LIN {X 0,Y 516.64,Z 251.361,A -85,B 0,C 180,E1 -4935.827,E2 -4935.827} C_VEL
LIN {X 0,Y 516.583,Z 256.504,A -85,B 0,C 180,E1 -4939.02,E2 -4939.02} C_VEL
LIN {X 0,Y 516.522,Z 261.674,A -85,B 0,C 180,E1 -4942.18,E2 -4942.18} C_VEL
LIN {X 0,Y 516.438,Z 265.584,A -85,B 0,C 180,E1 -4944.534,E2 -4944.534} C_VEL
LIN {X 0,Y 516.408,Z 269.551,A -85,B 0,C 180,E1 -4946.879,E2 -4946.879} C_VEL
LIN {X 0,Y 516.319,Z 273.421,A -85,B 0,C 180,E1 -4949.171,E2 -4949.171} C_VEL
LIN {X 0,Y 518.475,Z 285.209,A -85,B 0,C 180,E1 -4949.539,E2 -4949.539} C_VEL
LIN {X 0,Y 518.209,Z 297.677,A -85,B 0,C 180,E1 -4950,E2 -4950} C_VEL
LIN {X 0,Y 517.936,Z 309.297,A -85,B 0,C 180,E1 -4950.583,E2 -4950.583} C_VEL
LIN {X 0,Y 517.653,Z 319.894,A -85,B 0,C 180,E1 -4951.264,E2 -4951.264} C_VEL
LIN {X 0,Y 517.351,Z 330.743,A -85,B 0,C 180,E1 -4952.141,E2 -4952.141} C_VEL
LIN {X 0,Y 517.046,Z 340.474,A -85,B 0,C 180,E1 -4953.117,E2 -4953.117} C_VEL
LIN {X 0,Y 516.799,Z 348.474,A -85,B 0,C 180,E1 -4954.094,E2 -4954.094} C_VEL
LIN {X 0,Y 516.581,Z 356.35,A -85,B 0,C 180,E1 -4955.269,E2 -4955.269} C_VEL
LIN {X 0,Y 516.504,Z 361.681,A -85,B 0,C 180,E1 -4956.249,E2 -4956.249} C_VEL
LIN {X 0,Y 516.401,Z 366.925,A -85,B 0,C 180,E1 -4957.428,E2 -4957.428} C_VEL
LIN {X 0,Y 516.324,Z 371.016,A -85,B 0,C 180,E1 -4958.611,E2 -4958.611} C_VEL
LIN {X 0,Y 516.234,Z 373.162,A -85,B 0,C 180,E1 -4959.402,E2 -4959.402} C_VEL
LIN {X 0,Y 516.257,Z 374.841,A -85,B 0,C 180,E1 -4960.193,E2 -4960.193} C_VEL
LIN {X 0,Y 516.287,Z 376.666,A -85,B 0,C 180,E1 -4961.455,E2 -4961.455} C_VEL
LIN {X 0,Y 516.17,Z 377.425,A -85,B 0,C 180,E1 -4962.582,E2 -4962.582} C_VEL
LIN {X 0,Y 516.164,Z 377.451,A -85,B 0,C 180,E1 -4963.383,E2 -4963.383} C_VEL
LIN {X 0,Y 516.222,Z 376.448,A -85,B 0,C 180,E1 -4964.852,E2 -4964.852} C_VEL
LIN {X 0,Y 516.177,Z 375.022,A -85,B 0,C 180,E1 -4965.801,E2 -4965.801} C_VEL
LIN {X 0,Y 516.285,Z 372.314,A -85,B 0,C 180,E1 -4967.017,E2 -4967.017} C_VEL
LIN {X 0,Y 516.383,Z 368.5,A -85,B 0,C 180,E1 -4968.242,E2 -4968.242} C_VEL
LIN {X 0,Y 516.495,Z 363.45,A -85,B 0,C 180,E1 -4969.473,E2 -4969.473} C_VEL
LIN {X 0,Y 516.618,Z 356.988,A -85,B 0,C 180,E1 -4970.713,E2 -4970.713} C_VEL
LIN {X 0,Y 516.781,Z 350.287,A -85,B 0,C 180,E1 -4971.751,E2 -4971.751} C_VEL
LIN {X 0,Y 517.049,Z 341.465,A -85,B 0,C 180,E1 -4972.865,E2 -4972.865} C_VEL
LIN {X 0,Y 517.324,Z 331.971,A -85,B 0,C 180,E1 -4973.838,E2 -4973.838} C_VEL
LIN {X 0,Y 517.624,Z 320.871,A -85,B 0,C 180,E1 -4974.758,E2 -4974.758} C_VEL
LIN {X 0,Y 517.869,Z 310.954,A -85,B 0,C 180,E1 -4975.415,E2 -4975.415} C_VEL
LIN {X 0,Y 518.19,Z 300.085,A -85,B 0,C 180,E1 -4975.986,E2 -4975.986} C_VEL
LIN {X 0,Y 518.46,Z 287.154,A -85,B 0,C 180,E1 -4976.489,E2 -4976.489} C_VEL
LIN {X 0,Y 518.135,Z 283.054,A -85,B 0,C 180,E1 -4976.625,E2 -4976.625} C_VEL
LIN {X 0,Y 516.3,Z 273.441,A -85,B 0,C 180,E1 -4976.915,E2 -4976.915} C_VEL
LIN {X 0,Y 516.312,Z 269.236,A -85,B 0,C 180,E1 -4979.409,E2 -4979.409} C_VEL
LIN {X 0,Y 516.428,Z 264.137,A -85,B 0,C 180,E1 -4982.464,E2 -4982.464} C_VEL
LIN {X 0,Y 516.466,Z 259.546,A -85,B 0,C 180,E1 -4985.269,E2 -4985.269} C_VEL
LIN {X 0,Y 516.563,Z 255.307,A -85,B 0,C 180,E1 -4987.9,E2 -4987.9} C_VEL
LIN {X 0,Y 516.585,Z 250.785,A -85,B 0,C 180,E1 -4990.769,E2 -4990.769} C_VEL
LIN {X 0,Y 516.728,Z 245.918,A -85,B 0,C 180,E1 -4993.918,E2 -4993.918} C_VEL
LIN {X 0,Y 516.816,Z 242.592,A -85,B 0,C 180,E1 -4996.113,E2 -4996.113} C_VEL
LIN {X 0,Y 516.828,Z 239.255,A -85,B 0,C 180,E1 -4998.408,E2 -4998.408} C_VEL
LIN {X 0,Y 516.867,Z 239.107,A -85,B 0,C 180,E1 -5001.285,E2 -5001.285} C_VEL
LIN {X 0,Y 516.878,Z 239.105,A -85,B 0,C 180,E1 -5004.222,E2 -5004.222} C_VEL
LIN {X 0,Y 516.882,Z 239.104,A -85,B 0,C 180,E1 -5007.054,E2 -5007.054} C_VEL
LIN {X 0,Y 516.889,Z 239.099,A -85,B 0,C 180,E1 -5009.797,E2 -5009.797} C_VEL
LIN {X 0,Y 516.915,Z 239.095,A -85,B 0,C 180,E1 -5012.468,E2 -5012.468} C_VEL
LIN {X 0,Y 516.897,Z 239.1,A -85,B 0,C 180,E1 -5015.072,E2 -5015.072} C_VEL
LIN {X 0,Y 516.9,Z 239.098,A -85,B 0,C 180,E1 -5017.624,E2 -5017.624} C_VEL
LIN {X 0,Y 516.919,Z 239.094,A -85,B 0,C 180,E1 -5020.13,E2 -5020.13} C_VEL
LIN {X 0,Y 516.919,Z 239.097,A -85,B 0,C 180,E1 -5022.597,E2 -5022.597} C_VEL
LIN {X 0,Y 516.929,Z 239.094,A -85,B 0,C 180,E1 -5025.031,E2 -5025.031} C_VEL
LIN {X 0,Y 516.953,Z 239.093,A -85,B 0,C 180,E1 -5028.234,E2 -5028.234} C_VEL
LIN {X 0,Y 516.962,Z 239.094,A -85,B 0,C 180,E1 -5031.401,E2 -5031.401} C_VEL
LIN {X 0,Y 516.984,Z 239.086,A -85,B 0,C 180,E1 -5033.758,E2 -5033.758} C_VEL
LIN {X 0,Y 517.009,Z 239.083,A -85,B 0,C 180,E1 -5036.884,E2 -5036.884} C_VEL
LIN {X 0,Y 517.069,Z 239.076,A -85,B 0,C 180,E1 -5040.001,E2 -5040.001} C_VEL
LIN {X 0,Y 517.007,Z 239.085,A -85,B 0,C 180,E1 -5043.118,E2 -5043.118} C_VEL
LIN {X 0,Y 516.992,Z 239.087,A -85,B 0,C 180,E1 -5046.244,E2 -5046.244} C_VEL
LIN {X 0,Y 516.945,Z 239.095,A -85,B 0,C 180,E1 -5049.39,E2 -5049.39} C_VEL
LIN {X 0,Y 516.948,Z 239.09,A -85,B 0,C 180,E1 -5051.811,E2 -5051.811} C_VEL
LIN {X 0,Y 516.934,Z 239.094,A -85,B 0,C 180,E1 -5055.147,E2 -5055.147} C_VEL
LIN {X 0,Y 516.918,Z 239.097,A -85,B 0,C 180,E1 -5058.223,E2 -5058.223} C_VEL
LIN {X 0,Y 516.897,Z 239.099,A -85,B 0,C 180,E1 -5060.703,E2 -5060.703} C_VEL
LIN {X 0,Y 516.905,Z 239.098,A -85,B 0,C 180,E1 -5064.073,E2 -5064.073} C_VEL
LIN {X 0,Y 516.905,Z 239.099,A -85,B 0,C 180,E1 -5066.66,E2 -5066.66} C_VEL
LIN {X 0,Y 516.904,Z 239.099,A -85,B 0,C 180,E1 -5069.525,E2 -5069.525} C_VEL
LIN {X 0,Y 516.893,Z 239.1,A -85,B 0,C 180,E1 -5072.545,E2 -5072.545} C_VEL
LIN {X 0,Y 516.861,Z 239.106,A -85,B 0,C 180,E1 -5075.331,E2 -5075.331} C_VEL
LIN {X 0,Y 516.877,Z 239.102,A -85,B 0,C 180,E1 -5077.944,E2 -5077.944} C_VEL
LIN {X 0,Y 516.879,Z 239.098,A -85,B 0,C 180,E1 -5080.743,E2 -5080.743} C_VEL
LIN {X 0,Y 516.881,Z 239.103,A -85,B 0,C 180,E1 -5082.832,E2 -5082.832} C_VEL
LIN {X 0,Y 516.892,Z 239.096,A -85,B 0,C 180,E1 -5085.008,E2 -5085.008} C_VEL
LIN {X 0,Y 516.885,Z 239.103,A -85,B 0,C 180,E1 -5088.403,E2 -5088.403} C_VEL
LIN {X 0,Y 516.873,Z 239.106,A -85,B 0,C 180,E1 -5091.703,E2 -5091.703} C_VEL
LIN {X 0,Y 516.917,Z 239.169,A -85,B 0,C 180,E1 -5092.053,E2 -5092.053} C_VEL
LIN {X 0,Y 517.587,Z 243.814,A -85,B 0,C 180,E1 -5094.278,E2 -5094.278} C_VEL
LIN {X 0,Y 517.503,Z 249.096,A -85,B 0,C 180,E1 -5096.633,E2 -5096.633} C_VEL
LIN {X 0,Y 517.24,Z 255.558,A -85,B 0,C 180,E1 -5099.368,E2 -5099.368} C_VEL
LIN {X 0,Y 517.074,Z 262.165,A -85,B 0,C 180,E1 -5102.065,E2 -5102.065} C_VEL
LIN {X 0,Y 516.895,Z 269.812,A -85,B 0,C 180,E1 -5105.072,E2 -5105.072} C_VEL
LIN {X 0,Y 516.755,Z 277.613,A -85,B 0,C 180,E1 -5108.047,E2 -5108.047} C_VEL
LIN {X 0,Y 516.6,Z 285.437,A -85,B 0,C 180,E1 -5110.944,E2 -5110.944} C_VEL
LIN {X 0,Y 516.528,Z 293.29,A -85,B 0,C 180,E1 -5113.804,E2 -5113.804} C_VEL
LIN {X 0,Y 516.474,Z 299.682,A -85,B 0,C 180,E1 -5116.098,E2 -5116.098} C_VEL
LIN {X 0,Y 518.432,Z 313.107,A -85,B 0,C 180,E1 -5116.477,E2 -5116.477} C_VEL
LIN {X 0,Y 518.143,Z 326.44,A -85,B 0,C 180,E1 -5116.968,E2 -5116.968} C_VEL
LIN {X 0,Y 517.861,Z 337.809,A -85,B 0,C 180,E1 -5117.539,E2 -5117.539} C_VEL
LIN {X 0,Y 517.534,Z 348.854,A -85,B 0,C 180,E1 -5118.247,E2 -5118.247} C_VEL
LIN {X 0,Y 517.294,Z 359.775,A -85,B 0,C 180,E1 -5119.135,E2 -5119.135} C_VEL
LIN {X 0,Y 516.986,Z 368.678,A -85,B 0,C 180,E1 -5120.019,E2 -5120.019} C_VEL
LIN {X 0,Y 516.749,Z 378.354,A -85,B 0,C 180,E1 -5121.199,E2 -5121.199} C_VEL
LIN {X 0,Y 516.557,Z 386.057,A -85,B 0,C 180,E1 -5122.377,E2 -5122.377} C_VEL
LIN {X 0,Y 516.412,Z 393.157,A -85,B 0,C 180,E1 -5123.75,E2 -5123.75} C_VEL
LIN {X 0,Y 516.313,Z 397.88,A -85,B 0,C 180,E1 -5124.924,E2 -5124.924} C_VEL
LIN {X 0,Y 516.352,Z 401.492,A -85,B 0,C 180,E1 -5126.098,E2 -5126.098} C_VEL
LIN {X 0,Y 516.283,Z 403.352,A -85,B 0,C 180,E1 -5126.879,E2 -5126.879} C_VEL
LIN {X 0,Y 516.262,Z 404.748,A -85,B 0,C 180,E1 -5127.659,E2 -5127.659} C_VEL
LIN {X 0,Y 516.16,Z 406.35,A -85,B 0,C 180,E1 -5129.22,E2 -5129.22} C_VEL
LIN {X 0,Y 516.154,Z 406.567,A -85,B 0,C 180,E1 -5130,E2 -5130} C_VEL
LIN {X 0,Y 516.192,Z 405.747,A -85,B 0,C 180,E1 -5131.56,E2 -5131.56} C_VEL
LIN {X 0,Y 516.262,Z 404.755,A -85,B 0,C 180,E1 -5132.341,E2 -5132.341} C_VEL
LIN {X 0,Y 516.283,Z 403.361,A -85,B 0,C 180,E1 -5133.121,E2 -5133.121} C_VEL
LIN {X 0,Y 516.313,Z 400.427,A -85,B 0,C 180,E1 -5134.293,E2 -5134.293} C_VEL
LIN {X 0,Y 516.376,Z 396.456,A -85,B 0,C 180,E1 -5135.467,E2 -5135.467} C_VEL
LIN {X 0,Y 516.476,Z 390.586,A -85,B 0,C 180,E1 -5136.792,E2 -5136.792} C_VEL
LIN {X 0,Y 516.608,Z 383.672,A -85,B 0,C 180,E1 -5138.015,E2 -5138.015} C_VEL
LIN {X 0,Y 516.828,Z 375.389,A -85,B 0,C 180,E1 -5139.194,E2 -5139.194} C_VEL
LIN {X 0,Y 517.035,Z 366.898,A -85,B 0,C 180,E1 -5140.178,E2 -5140.178} C_VEL
LIN {X 0,Y 517.353,Z 356.407,A -85,B 0,C 180,E1 -5141.162,E2 -5141.162} C_VEL
LIN {X 0,Y 517.659,Z 345.383,A -85,B 0,C 180,E1 -5141.994,E2 -5141.994} C_VEL
LIN {X 0,Y 517.95,Z 334.655,A -85,B 0,C 180,E1 -5142.638,E2 -5142.638} C_VEL
LIN {X 0,Y 518.269,Z 322.988,A -85,B 0,C 180,E1 -5143.178,E2 -5143.178} C_VEL
LIN {X 0,Y 518.281,Z 311.371,A -85,B 0,C 180,E1 -5143.577,E2 -5143.577} C_VEL
LIN {X 0,Y 516.474,Z 299.725,A -85,B 0,C 180,E1 -5143.902,E2 -5143.902} C_VEL
LIN {X 0,Y 516.547,Z 291.102,A -85,B 0,C 180,E1 -5147.009,E2 -5147.009} C_VEL
LIN {X 0,Y 516.663,Z 283.255,A -85,B 0,C 180,E1 -5149.88,E2 -5149.88} C_VEL
LIN {X 0,Y 516.77,Z 275.434,A -85,B 0,C 180,E1 -5152.804,E2 -5152.804} C_VEL
LIN {X 0,Y 516.93,Z 268.729,A -85,B 0,C 180,E1 -5155.357,E2 -5155.357} C_VEL
LIN {X 0,Y 517.09,Z 260.925,A -85,B 0,C 180,E1 -5158.404,E2 -5158.404} C_VEL
LIN {X 0,Y 517.294,Z 253.129,A -85,B 0,C 180,E1 -5161.537,E2 -5161.537} C_VEL
LIN {X 0,Y 517.497,Z 247.024,A -85,B 0,C 180,E1 -5164.062,E2 -5164.062} C_VEL
LIN {X 0,Y 517.503,Z 243.125,A -85,B 0,C 180,E1 -5165.729,E2 -5165.729} C_VEL
LIN {X 0,Y 516.891,Z 239.102,A -85,B 0,C 180,E1 -5167.599,E2 -5167.599} C_VEL
LIN {X 0,Y 516.846,Z 239.108,A -85,B 0,C 180,E1 -5170.744,E2 -5170.744} C_VEL
LIN {X 0,Y 516.857,Z 239.099,A -85,B 0,C 180,E1 -5173.905,E2 -5173.905} C_VEL
LIN {X 0,Y 516.855,Z 239.101,A -85,B 0,C 180,E1 -5176.109,E2 -5176.109} C_VEL
LIN {X 0,Y 516.842,Z 239.102,A -85,B 0,C 180,E1 -5179.254,E2 -5179.254} C_VEL
LIN {X 0,Y 516.848,Z 239.104,A -85,B 0,C 180,E1 -5182.06,E2 -5182.06} C_VEL
LIN {X 0,Y 516.868,Z 239.098,A -85,B 0,C 180,E1 -5185.173,E2 -5185.173} C_VEL
LIN {X 0,Y 516.867,Z 239.103,A -85,B 0,C 180,E1 -5187.974,E2 -5187.974} C_VEL
LIN {X 0,Y 516.913,Z 239.094,A -85,B 0,C 180,E1 -5190.694,E2 -5190.694} C_VEL
LIN {X 0,Y 516.891,Z 239.101,A -85,B 0,C 180,E1 -5193.813,E2 -5193.813} C_VEL
LIN {X 0,Y 516.852,Z 239.101,A -85,B 0,C 180,E1 -5196.775,E2 -5196.775} C_VEL
LIN {X 0,Y 516.932,Z 239.096,A -85,B 0,C 180,E1 -5199.731,E2 -5199.731} C_VEL
LIN {X 0,Y 516.899,Z 239.095,A -85,B 0,C 180,E1 -5202.594,E2 -5202.594} C_VEL
LIN {X 0,Y 516.934,Z 239.094,A -85,B 0,C 180,E1 -5205.029,E2 -5205.029} C_VEL
LIN {X 0,Y 516.957,Z 239.088,A -85,B 0,C 180,E1 -5208.233,E2 -5208.233} C_VEL
LIN {X 0,Y 516.96,Z 239.093,A -85,B 0,C 180,E1 -5211.399,E2 -5211.399} C_VEL
LIN {X 0,Y 516.999,Z 239.084,A -85,B 0,C 180,E1 -5213.756,E2 -5213.756} C_VEL
LIN {X 0,Y 517.073,Z 239.074,A -85,B 0,C 180,E1 -5217.662,E2 -5217.662} C_VEL
LIN {X 0,Y 517.087,Z 239.076,A -85,B 0,C 180,E1 -5220.778,E2 -5220.778} C_VEL
LIN {X 0,Y 517.007,Z 239.084,A -85,B 0,C 180,E1 -5223.116,E2 -5223.116} C_VEL
LIN {X 0,Y 517,Z 239.087,A -85,B 0,C 180,E1 -5226.242,E2 -5226.242} C_VEL
LIN {X 0,Y 516.949,Z 239.089,A -85,B 0,C 180,E1 -5229.388,E2 -5229.388} C_VEL
LIN {X 0,Y 516.946,Z 239.092,A -85,B 0,C 180,E1 -5231.809,E2 -5231.809} C_VEL
LIN {X 0,Y 516.932,Z 239.091,A -85,B 0,C 180,E1 -5235.146,E2 -5235.146} C_VEL
LIN {X 0,Y 516.914,Z 239.097,A -85,B 0,C 180,E1 -5238.221,E2 -5238.221} C_VEL
LIN {X 0,Y 516.901,Z 239.095,A -85,B 0,C 180,E1 -5240.701,E2 -5240.701} C_VEL
LIN {X 0,Y 516.899,Z 239.098,A -85,B 0,C 180,E1 -5244.071,E2 -5244.071} C_VEL
LIN {X 0,Y 516.917,Z 239.092,A -85,B 0,C 180,E1 -5246.657,E2 -5246.657} C_VEL
LIN {X 0,Y 516.912,Z 239.099,A -85,B 0,C 180,E1 -5249.526,E2 -5249.526} C_VEL
LIN {X 0,Y 516.888,Z 239.096,A -85,B 0,C 180,E1 -5252.544,E2 -5252.544} C_VEL
LIN {X 0,Y 516.871,Z 239.104,A -85,B 0,C 180,E1 -5255.332,E2 -5255.332} C_VEL
LIN {X 0,Y 516.872,Z 239.097,A -85,B 0,C 180,E1 -5257.943,E2 -5257.943} C_VEL
LIN {X 0,Y 516.896,Z 239.098,A -85,B 0,C 180,E1 -5260.739,E2 -5260.739} C_VEL
LIN {X 0,Y 516.869,Z 239.097,A -85,B 0,C 180,E1 -5263.903,E2 -5263.903} C_VEL
LIN {X 0,Y 516.869,Z 239.098,A -85,B 0,C 180,E1 -5266.107,E2 -5266.107} C_VEL
LIN {X 0,Y 516.904,Z 239.097,A -85,B 0,C 180,E1 -5268.398,E2 -5268.398} C_VEL
LIN {X 0,Y 516.868,Z 239.101,A -85,B 0,C 180,E1 -5270.315,E2 -5270.315} C_VEL
LIN {X 0,Y 516.199,Z 239.185,A -85,B 0,C 180,E1 -5270.965,E2 -5270.965} C_VEL
LIN {X 0,Y 513.353,Z 239.537,A -85,B 0,C 180,E1 -5272.021,E2 -5272.021} C_VEL
LIN {X 0,Y 510.945,Z 239.839,A -85,B 0,C 180,E1 -5272.871,E2 -5272.871} C_VEL
LIN {X 0,Y 509.904,Z 239.965,A -85,B 0,C 180,E1 -5273.528,E2 -5273.528} C_VEL
LIN {X 0,Y 509.816,Z 239.977,A -85,B 0,C 180,E1 -5273.75,E2 -5273.75} C_VEL
LIN {X 0,Y 509.848,Z 239.978,A -85,B 0,C 180,E1 -5276.539,E2 -5276.539} C_VEL
LIN {X 0,Y 509.832,Z 239.974,A -85,B 0,C 180,E1 -5279.334,E2 -5279.334} C_VEL
LIN {X 0,Y 509.878,Z 239.975,A -85,B 0,C 180,E1 -5282.054,E2 -5282.054} C_VEL
LIN {X 0,Y 509.811,Z 239.978,A -85,B 0,C 180,E1 -5284.701,E2 -5284.701} C_VEL
LIN {X 0,Y 509.736,Z 239.99,A -85,B 0,C 180,E1 -5287.479,E2 -5287.479} C_VEL
LIN {X 0,Y 509.687,Z 240.157,A -85,B 0,C 180,E1 -5288.143,E2 -5288.143} C_VEL
LIN {X 0,Y 509.695,Z 244.024,A -85,B 0,C 180,E1 -5290.675,E2 -5290.675} C_VEL
LIN {X 0,Y 509.609,Z 247.895,A -85,B 0,C 180,E1 -5293.166,E2 -5293.166} C_VEL
LIN {X 0,Y 509.592,Z 251.768,A -85,B 0,C 180,E1 -5295.627,E2 -5295.627} C_VEL
LIN {X 0,Y 509.521,Z 256.934,A -85,B 0,C 180,E1 -5298.866,E2 -5298.866} C_VEL
LIN {X 0,Y 509.449,Z 262.123,A -85,B 0,C 180,E1 -5302.071,E2 -5302.071} C_VEL
LIN {X 0,Y 509.514,Z 264.724,A -85,B 0,C 180,E1 -5303.665,E2 -5303.665} C_VEL
LIN {X 0,Y 509.35,Z 270.009,A -85,B 0,C 180,E1 -5306.836,E2 -5306.836} C_VEL
LIN {X 0,Y 509.24,Z 273.729,A -85,B 0,C 180,E1 -5308.987,E2 -5308.987} C_VEL
LIN {X 0,Y 511.525,Z 285.655,A -85,B 0,C 180,E1 -5309.36,E2 -5309.36} C_VEL
LIN {X 0,Y 511.288,Z 298.579,A -85,B 0,C 180,E1 -5309.852,E2 -5309.852} C_VEL
LIN {X 0,Y 510.974,Z 310.903,A -85,B 0,C 180,E1 -5310.492,E2 -5310.492} C_VEL
LIN {X 0,Y 510.627,Z 322.466,A -85,B 0,C 180,E1 -5311.281,E2 -5311.281} C_VEL
LIN {X 0,Y 510.325,Z 332.859,A -85,B 0,C 180,E1 -5312.17,E2 -5312.17} C_VEL
LIN {X 0,Y 509.981,Z 342.279,A -85,B 0,C 180,E1 -5313.16,E2 -5313.16} C_VEL
LIN {X 0,Y 509.716,Z 351.352,A -85,B 0,C 180,E1 -5314.349,E2 -5314.349} C_VEL
LIN {X 0,Y 509.471,Z 358.687,A -85,B 0,C 180,E1 -5315.541,E2 -5315.541} C_VEL
LIN {X 0,Y 509.384,Z 365.171,A -85,B 0,C 180,E1 -5316.869,E2 -5316.869} C_VEL
LIN {X 0,Y 509.279,Z 370.533,A -85,B 0,C 180,E1 -5318.331,E2 -5318.331} C_VEL
LIN {X 0,Y 509.139,Z 373.77,A -85,B 0,C 180,E1 -5319.534,E2 -5319.534} C_VEL
LIN {X 0,Y 509.175,Z 375.372,A -85,B 0,C 180,E1 -5320.337,E2 -5320.337} C_VEL
LIN {X 0,Y 509.187,Z 376.927,A -85,B 0,C 180,E1 -5321.495,E2 -5321.495} C_VEL
LIN {X 0,Y 509.09,Z 377.661,A -85,B 0,C 180,E1 -5322.76,E2 -5322.76} C_VEL
LIN {X 0,Y 509.073,Z 377.613,A -85,B 0,C 180,E1 -5323.573,E2 -5323.573} C_VEL
LIN {X 0,Y 509.127,Z 376.597,A -85,B 0,C 180,E1 -5324.927,E2 -5324.927} C_VEL
LIN {X 0,Y 509.09,Z 374.881,A -85,B 0,C 180,E1 -5326.027,E2 -5326.027} C_VEL
LIN {X 0,Y 509.212,Z 372.012,A -85,B 0,C 180,E1 -5327.261,E2 -5327.261} C_VEL
LIN {X 0,Y 509.326,Z 368.025,A -85,B 0,C 180,E1 -5328.503,E2 -5328.503} C_VEL
LIN {X 0,Y 509.424,Z 362.784,A -85,B 0,C 180,E1 -5329.755,E2 -5329.755} C_VEL
LIN {X 0,Y 509.574,Z 356.049,A -85,B 0,C 180,E1 -5331.013,E2 -5331.013} C_VEL
LIN {X 0,Y 509.837,Z 347.76,A -85,B 0,C 180,E1 -5332.245,E2 -5332.245} C_VEL
LIN {X 0,Y 510.123,Z 338.713,A -85,B 0,C 180,E1 -5333.333,E2 -5333.333} C_VEL
LIN {X 0,Y 510.418,Z 328.858,A -85,B 0,C 180,E1 -5334.289,E2 -5334.289} C_VEL
LIN {X 0,Y 510.731,Z 317.571,A -85,B 0,C 180,E1 -5335.169,E2 -5335.169} C_VEL
LIN {X 0,Y 511.106,Z 305.865,A -85,B 0,C 180,E1 -5335.885,E2 -5335.885} C_VEL
LIN {X 0,Y 511.452,Z 293.198,A -85,B 0,C 180,E1 -5336.464,E2 -5336.464} C_VEL
LIN {X 0,Y 511.428,Z 285.138,A -85,B 0,C 180,E1 -5336.751,E2 -5336.751} C_VEL
LIN {X 0,Y 509.214,Z 273.634,A -85,B 0,C 180,E1 -5337.121,E2 -5337.121} C_VEL
LIN {X 0,Y 509.242,Z 269.172,A -85,B 0,C 180,E1 -5339.79,E2 -5339.79} C_VEL
LIN {X 0,Y 509.359,Z 264.397,A -85,B 0,C 180,E1 -5342.687,E2 -5342.687} C_VEL
LIN {X 0,Y 509.402,Z 259.835,A -85,B 0,C 180,E1 -5345.514,E2 -5345.514} C_VEL
LIN {X 0,Y 509.511,Z 255.307,A -85,B 0,C 180,E1 -5348.367,E2 -5348.367} C_VEL
LIN {X 0,Y 509.581,Z 249.896,A -85,B 0,C 180,E1 -5351.864,E2 -5351.864} C_VEL
LIN {X 0,Y 509.725,Z 245.622,A -85,B 0,C 180,E1 -5354.681,E2 -5354.681} C_VEL
LIN {X 0,Y 509.789,Z 241.504,A -85,B 0,C 180,E1 -5357.507,E2 -5357.507} C_VEL
LIN {X 0,Y 509.783,Z 239.989,A -85,B 0,C 180,E1 -5358.569,E2 -5358.569} C_VEL
LIN {X 0,Y 509.838,Z 239.978,A -85,B 0,C 180,E1 -5361.787,E2 -5361.787} C_VEL
LIN {X 0,Y 509.833,Z 239.98,A -85,B 0,C 180,E1 -5364.624,E2 -5364.624} C_VEL
LIN {X 0,Y 509.849,Z 239.98,A -85,B 0,C 180,E1 -5367.481,E2 -5367.481} C_VEL
LIN {X 0,Y 509.869,Z 239.978,A -85,B 0,C 180,E1 -5370.269,E2 -5370.269} C_VEL
LIN {X 0,Y 509.871,Z 239.974,A -85,B 0,C 180,E1 -5372.945,E2 -5372.945} C_VEL
LIN {X 0,Y 509.86,Z 239.974,A -85,B 0,C 180,E1 -5375.575,E2 -5375.575} C_VEL
LIN {X 0,Y 509.84,Z 239.978,A -85,B 0,C 180,E1 -5378.151,E2 -5378.151} C_VEL
LIN {X 0,Y 509.851,Z 239.977,A -85,B 0,C 180,E1 -5380.682,E2 -5380.682} C_VEL
LIN {X 0,Y 509.875,Z 239.971,A -85,B 0,C 180,E1 -5383.176,E2 -5383.176} C_VEL
LIN {X 0,Y 509.849,Z 239.977,A -85,B 0,C 180,E1 -5385.635,E2 -5385.635} C_VEL
LIN {X 0,Y 509.902,Z 239.969,A -85,B 0,C 180,E1 -5388.875,E2 -5388.875} C_VEL
LIN {X 0,Y 509.941,Z 239.964,A -85,B 0,C 180,E1 -5392.079,E2 -5392.079} C_VEL
LIN {X 0,Y 509.962,Z 239.966,A -85,B 0,C 180,E1 -5394.465,E2 -5394.465} C_VEL
LIN {X 0,Y 510.045,Z 239.954,A -85,B 0,C 180,E1 -5397.632,E2 -5397.632} C_VEL
LIN {X 0,Y 510.051,Z 239.952,A -85,B 0,C 180,E1 -5400.79,E2 -5400.79} C_VEL
LIN {X 0,Y 509.949,Z 239.964,A -85,B 0,C 180,E1 -5403.161,E2 -5403.161} C_VEL
LIN {X 0,Y 509.943,Z 239.966,A -85,B 0,C 180,E1 -5406.331,E2 -5406.331} C_VEL
LIN {X 0,Y 509.905,Z 239.968,A -85,B 0,C 180,E1 -5408.721,E2 -5408.721} C_VEL
LIN {X 0,Y 509.897,Z 239.969,A -85,B 0,C 180,E1 -5411.933,E2 -5411.933} C_VEL
LIN {X 0,Y 509.886,Z 239.973,A -85,B 0,C 180,E1 -5415.243,E2 -5415.243} C_VEL
LIN {X 0,Y 509.881,Z 239.973,A -85,B 0,C 180,E1 -5418.002,E2 -5418.002} C_VEL
LIN {X 0,Y 509.838,Z 239.978,A -85,B 0,C 180,E1 -5421.003,E2 -5421.003} C_VEL
LIN {X 0,Y 509.863,Z 239.978,A -85,B 0,C 180,E1 -5424.427,E2 -5424.427} C_VEL
LIN {X 0,Y 509.859,Z 239.976,A -85,B 0,C 180,E1 -5427.058,E2 -5427.058} C_VEL
LIN {X 0,Y 509.851,Z 239.977,A -85,B 0,C 180,E1 -5429.752,E2 -5429.752} C_VEL
LIN {X 0,Y 509.87,Z 239.974,A -85,B 0,C 180,E1 -5432.776,E2 -5432.776} C_VEL
LIN {X 0,Y 509.82,Z 239.98,A -85,B 0,C 180,E1 -5435.579,E2 -5435.579} C_VEL
LIN {X 0,Y 509.847,Z 239.979,A -85,B 0,C 180,E1 -5438.339,E2 -5438.339} C_VEL
LIN {X 0,Y 509.851,Z 239.978,A -85,B 0,C 180,E1 -5441.427,E2 -5441.427} C_VEL
LIN {X 0,Y 509.836,Z 239.975,A -85,B 0,C 180,E1 -5444.671,E2 -5444.671} C_VEL
LIN {X 0,Y 509.799,Z 239.987,A -85,B 0,C 180,E1 -5447.508,E2 -5447.508} C_VEL
LIN {X 0,Y 509.839,Z 239.981,A -85,B 0,C 180,E1 -5450.648,E2 -5450.648} C_VEL
LIN {X 0,Y 509.858,Z 239.981,A -85,B 0,C 180,E1 -5451.786,E2 -5451.786} C_VEL
LIN {X 0,Y 510.598,Z 245.135,A -85,B 0,C 180,E1 -5454.301,E2 -5454.301} C_VEL
LIN {X 0,Y 510.522,Z 250.211,A -85,B 0,C 180,E1 -5456.589,E2 -5456.589} C_VEL
LIN {X 0,Y 510.238,Z 256.623,A -85,B 0,C 180,E1 -5459.361,E2 -5459.361} C_VEL
LIN {X 0,Y 510.038,Z 263.137,A -85,B 0,C 180,E1 -5462.064,E2 -5462.064} C_VEL
LIN {X 0,Y 509.868,Z 269.723,A -85,B 0,C 180,E1 -5464.704,E2 -5464.704} C_VEL
LIN {X 0,Y 509.724,Z 276.866,A -85,B 0,C 180,E1 -5467.487,E2 -5467.487} C_VEL
LIN {X 0,Y 509.571,Z 284.152,A -85,B 0,C 180,E1 -5470.251,E2 -5470.251} C_VEL
LIN {X 0,Y 509.462,Z 291.989,A -85,B 0,C 180,E1 -5473.161,E2 -5473.161} C_VEL
LIN {X 0,Y 509.375,Z 299.472,A -85,B 0,C 180,E1 -5475.901,E2 -5475.901} C_VEL
LIN {X 0,Y 511.502,Z 313.659,A -85,B 0,C 180,E1 -5476.315,E2 -5476.315} C_VEL
LIN {X 0,Y 511.235,Z 326.228,A -85,B 0,C 180,E1 -5476.789,E2 -5476.789} C_VEL
LIN {X 0,Y 510.931,Z 337.623,A -85,B 0,C 180,E1 -5477.368,E2 -5477.368} C_VEL
LIN {X 0,Y 510.557,Z 348.643,A -85,B 0,C 180,E1 -5478.084,E2 -5478.084} C_VEL
LIN {X 0,Y 510.294,Z 359.565,A -85,B 0,C 180,E1 -5478.984,E2 -5478.984} C_VEL
LIN {X 0,Y 509.958,Z 368.469,A -85,B 0,C 180,E1 -5479.88,E2 -5479.88} C_VEL
LIN {X 0,Y 509.696,Z 378.147,A -85,B 0,C 180,E1 -5481.076,E2 -5481.076} C_VEL
LIN {X 0,Y 509.488,Z 385.851,A -85,B 0,C 180,E1 -5482.271,E2 -5482.271} C_VEL
LIN {X 0,Y 509.328,Z 392.05,A -85,B 0,C 180,E1 -5483.465,E2 -5483.465} C_VEL
LIN {X 0,Y 509.244,Z 397.678,A -85,B 0,C 180,E1 -5484.853,E2 -5484.853} C_VEL
LIN {X 0,Y 509.246,Z 401.289,A -85,B 0,C 180,E1 -5486.043,E2 -5486.043} C_VEL
LIN {X 0,Y 509.201,Z 403.151,A -85,B 0,C 180,E1 -5486.835,E2 -5486.835} C_VEL
LIN {X 0,Y 509.19,Z 404.548,A -85,B 0,C 180,E1 -5487.627,E2 -5487.627} C_VEL
LIN {X 0,Y 509.074,Z 406.151,A -85,B 0,C 180,E1 -5489.209,E2 -5489.209} C_VEL
LIN {X 0,Y 509.066,Z 406.368,A -85,B 0,C 180,E1 -5490,E2 -5490} C_VEL
LIN {X 0,Y 509.113,Z 405.548,A -85,B 0,C 180,E1 -5491.582,E2 -5491.582} C_VEL
LIN {X 0,Y 509.19,Z 404.556,A -85,B 0,C 180,E1 -5492.373,E2 -5492.373} C_VEL
LIN {X 0,Y 509.201,Z 403.162,A -85,B 0,C 180,E1 -5493.165,E2 -5493.165} C_VEL
LIN {X 0,Y 509.205,Z 400.227,A -85,B 0,C 180,E1 -5494.353,E2 -5494.353} C_VEL
LIN {X 0,Y 509.294,Z 396.257,A -85,B 0,C 180,E1 -5495.543,E2 -5495.543} C_VEL
LIN {X 0,Y 509.409,Z 390.249,A -85,B 0,C 180,E1 -5496.914,E2 -5496.914} C_VEL
LIN {X 0,Y 509.552,Z 383.471,A -85,B 0,C 180,E1 -5498.127,E2 -5498.127} C_VEL
LIN {X 0,Y 509.775,Z 375.187,A -85,B 0,C 180,E1 -5499.322,E2 -5499.322} C_VEL
LIN {X 0,Y 510.019,Z 366.696,A -85,B 0,C 180,E1 -5500.319,E2 -5500.319} C_VEL
LIN {X 0,Y 510.351,Z 356.205,A -85,B 0,C 180,E1 -5501.317,E2 -5501.317} C_VEL
LIN {X 0,Y 510.665,Z 345.179,A -85,B 0,C 180,E1 -5502.161,E2 -5502.161} C_VEL
LIN {X 0,Y 511.013,Z 334.452,A -85,B 0,C 180,E1 -5502.813,E2 -5502.813} C_VEL
LIN {X 0,Y 511.33,Z 322.782,A -85,B 0,C 180,E1 -5503.36,E2 -5503.36} C_VEL
LIN {X 0,Y 511.367,Z 312.081,A -85,B 0,C 180,E1 -5503.739,E2 -5503.739} C_VEL
LIN {X 0,Y 509.375,Z 299.524,A -85,B 0,C 180,E1 -5504.099,E2 -5504.099} C_VEL
LIN {X 0,Y 509.487,Z 290.937,A -85,B 0,C 180,E1 -5507.252,E2 -5507.252} C_VEL
LIN {X 0,Y 509.612,Z 282.713,A -85,B 0,C 180,E1 -5510.317,E2 -5510.317} C_VEL
LIN {X 0,Y 509.742,Z 275.289,A -85,B 0,C 180,E1 -5513.137,E2 -5513.137} C_VEL
LIN {X 0,Y 509.963,Z 267.48,A -85,B 0,C 180,E1 -5516.167,E2 -5516.167} C_VEL
LIN {X 0,Y 510.113,Z 259.668,A -85,B 0,C 180,E1 -5519.28,E2 -5519.28} C_VEL
LIN {X 0,Y 510.333,Z 251.875,A -85,B 0,C 180,E1 -5522.485,E2 -5522.485} C_VEL
LIN {X 0,Y 510.5,Z 245.205,A -85,B 0,C 180,E1 -5525.324,E2 -5525.324} C_VEL
LIN {X 0,Y 509.885,Z 240.201,A -85,B 0,C 180,E1 -5527.583,E2 -5527.583} C_VEL
LIN {X 0,Y 509.847,Z 239.978,A -85,B 0,C 180,E1 -5528.337,E2 -5528.337} C_VEL
LIN {X 0,Y 509.8,Z 239.981,A -85,B 0,C 180,E1 -5531.43,E2 -5531.43} C_VEL
LIN {X 0,Y 509.831,Z 239.98,A -85,B 0,C 180,E1 -5534.669,E2 -5534.669} C_VEL
LIN {X 0,Y 509.781,Z 239.981,A -85,B 0,C 180,E1 -5537.504,E2 -5537.504} C_VEL
LIN {X 0,Y 509.821,Z 239.983,A -85,B 0,C 180,E1 -5540.644,E2 -5540.644} C_VEL
LIN {X 0,Y 509.761,Z 239.984,A -85,B 0,C 180,E1 -5543.641,E2 -5543.641} C_VEL
LIN {X 0,Y 509.841,Z 239.978,A -85,B 0,C 180,E1 -5546.537,E2 -5546.537} C_VEL
LIN {X 0,Y 509.834,Z 239.975,A -85,B 0,C 180,E1 -5549.333,E2 -5549.333} C_VEL
LIN {X 0,Y 509.832,Z 239.981,A -85,B 0,C 180,E1 -5552.05,E2 -5552.05} C_VEL
LIN {X 0,Y 509.811,Z 239.978,A -85,B 0,C 180,E1 -5554.7,E2 -5554.7} C_VEL
LIN {X 0,Y 509.819,Z 239.981,A -85,B 0,C 180,E1 -5557.457,E2 -5557.457} C_VEL
LIN {X 0,Y 509.909,Z 239.972,A -85,B 0,C 180,E1 -5559.844,E2 -5559.844} C_VEL
LIN {X 0,Y 509.867,Z 239.975,A -85,B 0,C 180,E1 -5563.173,E2 -5563.173} C_VEL
LIN {X 0,Y 509.855,Z 239.978,A -85,B 0,C 180,E1 -5565.633,E2 -5565.633} C_VEL
LIN {X 0,Y 509.904,Z 239.97,A -85,B 0,C 180,E1 -5568.873,E2 -5568.873} C_VEL
LIN {X 0,Y 509.942,Z 239.962,A -85,B 0,C 180,E1 -5572.077,E2 -5572.077} C_VEL
LIN {X 0,Y 509.972,Z 239.96,A -85,B 0,C 180,E1 -5574.463,E2 -5574.463} C_VEL
LIN {X 0,Y 510.044,Z 239.95,A -85,B 0,C 180,E1 -5577.63,E2 -5577.63} C_VEL
LIN {X 0,Y 510.057,Z 239.952,A -85,B 0,C 180,E1 -5580.789,E2 -5580.789} C_VEL
LIN {X 0,Y 509.95,Z 239.963,A -85,B 0,C 180,E1 -5583.159,E2 -5583.159} C_VEL
LIN {X 0,Y 509.968,Z 239.964,A -85,B 0,C 180,E1 -5586.329,E2 -5586.329} C_VEL
LIN {X 0,Y 509.909,Z 239.97,A -85,B 0,C 180,E1 -5588.719,E2 -5588.719} C_VEL
LIN {X 0,Y 509.894,Z 239.971,A -85,B 0,C 180,E1 -5591.931,E2 -5591.931} C_VEL
LIN {X 0,Y 509.882,Z 239.969,A -85,B 0,C 180,E1 -5595.241,E2 -5595.241} C_VEL
LIN {X 0,Y 509.877,Z 239.975,A -85,B 0,C 180,E1 -5598,E2 -5598} C_VEL
LIN {X 0,Y 509.839,Z 239.974,A -85,B 0,C 180,E1 -5601.001,E2 -5601.001} C_VEL
LIN {X 0,Y 509.824,Z 239.981,A -85,B 0,C 180,E1 -5603.562,E2 -5603.562} C_VEL
LIN {X 0,Y 509.901,Z 239.967,A -85,B 0,C 180,E1 -5606.379,E2 -5606.379} C_VEL
LIN {X 0,Y 509.873,Z 239.97,A -85,B 0,C 180,E1 -5608.843,E2 -5608.843} C_VEL
LIN {X 0,Y 509.814,Z 239.982,A -85,B 0,C 180,E1 -5611.589,E2 -5611.589} C_VEL
LIN {X 0,Y 509.842,Z 239.973,A -85,B 0,C 180,E1 -5614.413,E2 -5614.413} C_VEL
LIN {X 0,Y 509.81,Z 239.982,A -85,B 0,C 180,E1 -5617.34,E2 -5617.34} C_VEL
LIN {X 0,Y 509.85,Z 239.973,A -85,B 0,C 180,E1 -5620.379,E2 -5620.379} C_VEL
LIN {X 0,Y 509.828,Z 239.981,A -85,B 0,C 180,E1 -5623.064,E2 -5623.064} C_VEL
LIN {X 0,Y 509.817,Z 239.975,A -85,B 0,C 180,E1 -5625.792,E2 -5625.792} C_VEL
LIN {X 0,Y 509.845,Z 239.978,A -85,B 0,C 180,E1 -5628.575,E2 -5628.575} C_VEL
LIN {X 0,Y 509.838,Z 239.973,A -85,B 0,C 180,E1 -5631.786,E2 -5631.786} C_VEL
LIN {X 0,Y 509.816,Z 239.977,A -85,B 0,C 180,E1 -5633.75,E2 -5633.75} C_VEL
LIN {X 0,Y 509.15,Z 240.066,A -85,B 0,C 180,E1 -5634.41,E2 -5634.41} C_VEL
LIN {X 0,Y 506.333,Z 240.414,A -85,B 0,C 180,E1 -5635.482,E2 -5635.482} C_VEL
LIN {X 0,Y 503.941,Z 240.715,A -85,B 0,C 180,E1 -5636.345,E2 -5636.345} C_VEL
LIN {X 0,Y 502.892,Z 240.84,A -85,B 0,C 180,E1 -5637.011,E2 -5637.011} C_VEL
LIN {X 0,Y 502.794,Z 240.851,A -85,B 0,C 180,E1 -5637.237,E2 -5637.237} C_VEL
LIN {X 0,Y 502.802,Z 240.855,A -85,B 0,C 180,E1 -5640.065,E2 -5640.065} C_VEL
LIN {X 0,Y 502.814,Z 240.852,A -85,B 0,C 180,E1 -5642.533,E2 -5642.533} C_VEL
LIN {X 0,Y 502.771,Z 240.855,A -85,B 0,C 180,E1 -5645.31,E2 -5645.31} C_VEL
LIN {X 0,Y 502.673,Z 240.872,A -85,B 0,C 180,E1 -5647.822,E2 -5647.822} C_VEL
LIN {X 0,Y 502.657,Z 243.102,A -85,B 0,C 180,E1 -5649.541,E2 -5649.541} C_VEL
LIN {X 0,Y 502.62,Z 246.983,A -85,B 0,C 180,E1 -5652.085,E2 -5652.085} C_VEL
LIN {X 0,Y 502.555,Z 252.162,A -85,B 0,C 180,E1 -5655.421,E2 -5655.421} C_VEL
LIN {X 0,Y 502.471,Z 257.348,A -85,B 0,C 180,E1 -5658.708,E2 -5658.708} C_VEL
LIN {X 0,Y 502.392,Z 262.568,A -85,B 0,C 180,E1 -5661.959,E2 -5661.959} C_VEL
LIN {X 0,Y 502.443,Z 265.187,A -85,B 0,C 180,E1 -5663.575,E2 -5663.575} C_VEL
LIN {X 0,Y 502.293,Z 270.466,A -85,B 0,C 180,E1 -5666.792,E2 -5666.792} C_VEL
LIN {X 0,Y 502.167,Z 273.779,A -85,B 0,C 180,E1 -5668.772,E2 -5668.772} C_VEL
LIN {X 0,Y 504.639,Z 286.79,A -85,B 0,C 180,E1 -5669.202,E2 -5669.202} C_VEL
LIN {X 0,Y 504.355,Z 299.49,A -85,B 0,C 180,E1 -5669.701,E2 -5669.701} C_VEL
LIN {X 0,Y 504.049,Z 310.8,A -85,B 0,C 180,E1 -5670.3,E2 -5670.3} C_VEL
LIN {X 0,Y 503.681,Z 322.434,A -85,B 0,C 180,E1 -5671.099,E2 -5671.099} C_VEL
LIN {X 0,Y 503.333,Z 332.873,A -85,B 0,C 180,E1 -5672,E2 -5672} C_VEL
LIN {X 0,Y 502.987,Z 342.32,A -85,B 0,C 180,E1 -5673.003,E2 -5673.003} C_VEL
LIN {X 0,Y 502.673,Z 351.434,A -85,B 0,C 180,E1 -5674.209,E2 -5674.209} C_VEL
LIN {X 0,Y 502.409,Z 358.789,A -85,B 0,C 180,E1 -5675.418,E2 -5675.418} C_VEL
LIN {X 0,Y 502.328,Z 365.561,A -85,B 0,C 180,E1 -5676.829,E2 -5676.829} C_VEL
LIN {X 0,Y 502.209,Z 370.054,A -85,B 0,C 180,E1 -5678.044,E2 -5678.044} C_VEL
LIN {X 0,Y 502.125,Z 372.43,A -85,B 0,C 180,E1 -5678.856,E2 -5678.856} C_VEL
LIN {X 0,Y 502.05,Z 374.378,A -85,B 0,C 180,E1 -5679.67,E2 -5679.67} C_VEL
LIN {X 0,Y 502.08,Z 375.895,A -85,B 0,C 180,E1 -5680.484,E2 -5680.484} C_VEL
LIN {X 0,Y 502.105,Z 377.197,A -85,B 0,C 180,E1 -5681.545,E2 -5681.545} C_VEL
LIN {X 0,Y 501.986,Z 377.899,A -85,B 0,C 180,E1 -5682.944,E2 -5682.944} C_VEL
LIN {X 0,Y 501.998,Z 377.746,A -85,B 0,C 180,E1 -5683.768,E2 -5683.768} C_VEL
LIN {X 0,Y 502.027,Z 376.742,A -85,B 0,C 180,E1 -5685.001,E2 -5685.001} C_VEL
LIN {X 0,Y 502.029,Z 374.735,A -85,B 0,C 180,E1 -5686.259,E2 -5686.259} C_VEL
LIN {X 0,Y 502.142,Z 371.746,A -85,B 0,C 180,E1 -5687.497,E2 -5687.497} C_VEL
LIN {X 0,Y 502.26,Z 367.525,A -85,B 0,C 180,E1 -5688.773,E2 -5688.773} C_VEL
LIN {X 0,Y 502.363,Z 362.188,A -85,B 0,C 180,E1 -5690.015,E2 -5690.015} C_VEL
LIN {X 0,Y 502.588,Z 355.07,A -85,B 0,C 180,E1 -5691.319,E2 -5691.319} C_VEL
LIN {X 0,Y 502.856,Z 347.134,A -85,B 0,C 180,E1 -5692.488,E2 -5692.488} C_VEL
LIN {X 0,Y 503.139,Z 338.074,A -85,B 0,C 180,E1 -5693.568,E2 -5693.568} C_VEL
LIN {X 0,Y 503.491,Z 328.029,A -85,B 0,C 180,E1 -5694.535,E2 -5694.535} C_VEL
LIN {X 0,Y 503.86,Z 316.717,A -85,B 0,C 180,E1 -5695.412,E2 -5695.412} C_VEL
LIN {X 0,Y 504.197,Z 304.31,A -85,B 0,C 180,E1 -5696.156,E2 -5696.156} C_VEL
LIN {X 0,Y 504.581,Z 291.848,A -85,B 0,C 180,E1 -5696.711,E2 -5696.711} C_VEL
LIN {X 0,Y 504.475,Z 285.815,A -85,B 0,C 180,E1 -5696.928,E2 -5696.928} C_VEL
LIN {X 0,Y 502.145,Z 273.811,A -85,B 0,C 180,E1 -5697.326,E2 -5697.326} C_VEL
LIN {X 0,Y 502.177,Z 268.99,A -85,B 0,C 180,E1 -5700.252,E2 -5700.252} C_VEL
LIN {X 0,Y 502.295,Z 264.419,A -85,B 0,C 180,E1 -5703.07,E2 -5703.07} C_VEL
LIN {X 0,Y 502.336,Z 259.786,A -85,B 0,C 180,E1 -5705.986,E2 -5705.986} C_VEL
LIN {X 0,Y 502.447,Z 255.071,A -85,B 0,C 180,E1 -5709.008,E2 -5709.008} C_VEL
LIN {X 0,Y 502.551,Z 250.262,A -85,B 0,C 180,E1 -5712.169,E2 -5712.169} C_VEL
LIN {X 0,Y 502.732,Z 245.361,A -85,B 0,C 180,E1 -5715.475,E2 -5715.475} C_VEL
LIN {X 0,Y 502.75,Z 241.938,A -85,B 0,C 180,E1 -5717.858,E2 -5717.858} C_VEL
LIN {X 0,Y 502.75,Z 240.864,A -85,B 0,C 180,E1 -5719.013,E2 -5719.013} C_VEL
LIN {X 0,Y 502.781,Z 240.857,A -85,B 0,C 180,E1 -5722.047,E2 -5722.047} C_VEL
LIN {X 0,Y 502.796,Z 240.855,A -85,B 0,C 180,E1 -5725.036,E2 -5725.036} C_VEL
LIN {X 0,Y 502.772,Z 240.858,A -85,B 0,C 180,E1 -5727.916,E2 -5727.916} C_VEL
LIN {X 0,Y 502.826,Z 240.851,A -85,B 0,C 180,E1 -5730.714,E2 -5730.714} C_VEL
LIN {X 0,Y 502.849,Z 240.851,A -85,B 0,C 180,E1 -5733.44,E2 -5733.44} C_VEL
LIN {X 0,Y 502.79,Z 240.857,A -85,B 0,C 180,E1 -5736.087,E2 -5736.087} C_VEL
LIN {X 0,Y 502.786,Z 240.855,A -85,B 0,C 180,E1 -5738.69,E2 -5738.69} C_VEL
LIN {X 0,Y 502.833,Z 240.849,A -85,B 0,C 180,E1 -5741.879,E2 -5741.879} C_VEL
LIN {X 0,Y 502.827,Z 240.849,A -85,B 0,C 180,E1 -5744.663,E2 -5744.663} C_VEL
LIN {X 0,Y 502.864,Z 240.846,A -85,B 0,C 180,E1 -5748.04,E2 -5748.04} C_VEL
LIN {X 0,Y 502.867,Z 240.847,A -85,B 0,C 180,E1 -5751.158,E2 -5751.158} C_VEL
LIN {X 0,Y 502.89,Z 240.841,A -85,B 0,C 180,E1 -5753.582,E2 -5753.582} C_VEL
LIN {X 0,Y 502.895,Z 240.842,A -85,B 0,C 180,E1 -5756.796,E2 -5756.796} C_VEL
LIN {X 0,Y 503.024,Z 240.827,A -85,B 0,C 180,E1 -5759.2,E2 -5759.2} C_VEL
LIN {X 0,Y 503.018,Z 240.827,A -85,B 0,C 180,E1 -5762.403,E2 -5762.403} C_VEL
LIN {X 0,Y 502.923,Z 240.837,A -85,B 0,C 180,E1 -5765.615,E2 -5765.615} C_VEL
LIN {X 0,Y 502.892,Z 240.846,A -85,B 0,C 180,E1 -5768.034,E2 -5768.034} C_VEL
LIN {X 0,Y 502.873,Z 240.846,A -85,B 0,C 180,E1 -5771.284,E2 -5771.284} C_VEL
LIN {X 0,Y 502.834,Z 240.85,A -85,B 0,C 180,E1 -5774.572,E2 -5774.572} C_VEL
LIN {X 0,Y 502.854,Z 240.848,A -85,B 0,C 180,E1 -5777.908,E2 -5777.908} C_VEL
LIN {X 0,Y 502.822,Z 240.853,A -85,B 0,C 180,E1 -5780.537,E2 -5780.537} C_VEL
LIN {X 0,Y 502.787,Z 240.86,A -85,B 0,C 180,E1 -5783.042,E2 -5783.042} C_VEL
LIN {X 0,Y 502.832,Z 240.852,A -85,B 0,C 180,E1 -5785.677,E2 -5785.677} C_VEL
LIN {X 0,Y 502.79,Z 240.856,A -85,B 0,C 180,E1 -5788.377,E2 -5788.377} C_VEL
LIN {X 0,Y 502.792,Z 240.856,A -85,B 0,C 180,E1 -5791.144,E2 -5791.144} C_VEL
LIN {X 0,Y 502.798,Z 240.856,A -85,B 0,C 180,E1 -5793.995,E2 -5793.995} C_VEL
LIN {X 0,Y 502.773,Z 240.857,A -85,B 0,C 180,E1 -5797.179,E2 -5797.179} C_VEL
LIN {X 0,Y 502.784,Z 240.855,A -85,B 0,C 180,E1 -5800.016,E2 -5800.016} C_VEL
LIN {X 0,Y 502.8,Z 240.853,A -85,B 0,C 180,E1 -5802.2,E2 -5802.2} C_VEL
LIN {X 0,Y 502.783,Z 240.855,A -85,B 0,C 180,E1 -5805.471,E2 -5805.471} C_VEL
LIN {X 0,Y 502.772,Z 240.862,A -85,B 0,C 180,E1 -5808.931,E2 -5808.931} C_VEL
LIN {X 0,Y 502.818,Z 240.93,A -85,B 0,C 180,E1 -5811.582,E2 -5811.582} C_VEL
LIN {X 0,Y 503.594,Z 246.006,A -85,B 0,C 180,E1 -5814.118,E2 -5814.118} C_VEL
LIN {X 0,Y 503.575,Z 250.21,A -85,B 0,C 180,E1 -5816.066,E2 -5816.066} C_VEL
LIN {X 0,Y 503.265,Z 256.594,A -85,B 0,C 180,E1 -5818.89,E2 -5818.89} C_VEL
LIN {X 0,Y 503.036,Z 263.151,A -85,B 0,C 180,E1 -5821.665,E2 -5821.665} C_VEL
LIN {X 0,Y 502.826,Z 270.741,A -85,B 0,C 180,E1 -5824.768,E2 -5824.768} C_VEL
LIN {X 0,Y 502.637,Z 278.462,A -85,B 0,C 180,E1 -5827.82,E2 -5827.82} C_VEL
LIN {X 0,Y 502.479,Z 286.235,A -85,B 0,C 180,E1 -5830.811,E2 -5830.811} C_VEL
LIN {X 0,Y 502.368,Z 294.044,A -85,B 0,C 180,E1 -5833.752,E2 -5833.752} C_VEL
LIN {X 0,Y 502.323,Z 299.513,A -85,B 0,C 180,E1 -5835.712,E2 -5835.712} C_VEL
LIN {X 0,Y 504.372,Z 312.673,A -85,B 0,C 180,E1 -5836.092,E2 -5836.092} C_VEL
LIN {X 0,Y 504.438,Z 322.541,A -85,B 0,C 180,E1 -5836.454,E2 -5836.454} C_VEL
LIN {X 0,Y 504.037,Z 334.204,A -85,B 0,C 180,E1 -5837.007,E2 -5837.007} C_VEL
LIN {X 0,Y 503.602,Z 346.288,A -85,B 0,C 180,E1 -5837.764,E2 -5837.764} C_VEL
LIN {X 0,Y 503.328,Z 357.141,A -85,B 0,C 180,E1 -5838.625,E2 -5838.625} C_VEL
LIN {X 0,Y 503,Z 366.459,A -85,B 0,C 180,E1 -5839.535,E2 -5839.535} C_VEL
LIN {X 0,Y 502.736,Z 374.955,A -85,B 0,C 180,E1 -5840.546,E2 -5840.546} C_VEL
LIN {X 0,Y 502.483,Z 383.244,A -85,B 0,C 180,E1 -5841.758,E2 -5841.758} C_VEL
LIN {X 0,Y 502.346,Z 389.928,A -85,B 0,C 180,E1 -5842.969,E2 -5842.969} C_VEL
LIN {X 0,Y 502.212,Z 396.042,A -85,B 0,C 180,E1 -5844.379,E2 -5844.379} C_VEL
LIN {X 0,Y 502.103,Z 400.014,A -85,B 0,C 180,E1 -5845.585,E2 -5845.585} C_VEL
LIN {X 0,Y 502.121,Z 402.95,A -85,B 0,C 180,E1 -5846.791,E2 -5846.791} C_VEL
LIN {X 0,Y 502.092,Z 404.347,A -85,B 0,C 180,E1 -5847.593,E2 -5847.593} C_VEL
LIN {X 0,Y 501.991,Z 405.951,A -85,B 0,C 180,E1 -5849.198,E2 -5849.198} C_VEL
LIN {X 0,Y 501.98,Z 406.168,A -85,B 0,C 180,E1 -5850,E2 -5850} C_VEL
LIN {X 0,Y 502.037,Z 405.349,A -85,B 0,C 180,E1 -5851.604,E2 -5851.604} C_VEL
LIN {X 0,Y 502.092,Z 404.357,A -85,B 0,C 180,E1 -5852.407,E2 -5852.407} C_VEL
LIN {X 0,Y 502.121,Z 402.963,A -85,B 0,C 180,E1 -5853.209,E2 -5853.209} C_VEL
LIN {X 0,Y 502.103,Z 400.028,A -85,B 0,C 180,E1 -5854.415,E2 -5854.415} C_VEL
LIN {X 0,Y 502.212,Z 396.057,A -85,B 0,C 180,E1 -5855.622,E2 -5855.622} C_VEL
LIN {X 0,Y 502.334,Z 390.049,A -85,B 0,C 180,E1 -5857.011,E2 -5857.011} C_VEL
LIN {X 0,Y 502.483,Z 383.27,A -85,B 0,C 180,E1 -5858.242,E2 -5858.242} C_VEL
LIN {X 0,Y 502.736,Z 374.986,A -85,B 0,C 180,E1 -5859.454,E2 -5859.454} C_VEL
LIN {X 0,Y 503.011,Z 366.494,A -85,B 0,C 180,E1 -5860.465,E2 -5860.465} C_VEL
LIN {X 0,Y 503.382,Z 356.003,A -85,B 0,C 180,E1 -5861.475,E2 -5861.475} C_VEL
LIN {X 0,Y 503.683,Z 344.975,A -85,B 0,C 180,E1 -5862.332,E2 -5862.332} C_VEL
LIN {X 0,Y 504.082,Z 334.249,A -85,B 0,C 180,E1 -5862.992,E2 -5862.992} C_VEL
LIN {X 0,Y 504.406,Z 322.577,A -85,B 0,C 180,E1 -5863.547,E2 -5863.547} C_VEL
LIN {X 0,Y 504.407,Z 312.716,A -85,B 0,C 180,E1 -5863.907,E2 -5863.907} C_VEL
LIN {X 0,Y 502.294,Z 299.328,A -85,B 0,C 180,E1 -5864.302,E2 -5864.302} C_VEL
LIN {X 0,Y 502.409,Z 290.766,A -85,B 0,C 180,E1 -5867.503,E2 -5867.503} C_VEL
LIN {X 0,Y 502.55,Z 282.954,A -85,B 0,C 180,E1 -5870.463,E2 -5870.463} C_VEL
LIN {X 0,Y 502.696,Z 275.136,A -85,B 0,C 180,E1 -5873.481,E2 -5873.481} C_VEL
LIN {X 0,Y 502.92,Z 267.303,A -85,B 0,C 180,E1 -5876.572,E2 -5876.572} C_VEL
LIN {X 0,Y 503.089,Z 260.636,A -85,B 0,C 180,E1 -5879.27,E2 -5879.27} C_VEL
LIN {X 0,Y 503.313,Z 252.838,A -85,B 0,C 180,E1 -5882.519,E2 -5882.519} C_VEL
LIN {X 0,Y 503.485,Z 246.163,A -85,B 0,C 180,E1 -5885.399,E2 -5885.399} C_VEL
LIN {X 0,Y 502.923,Z 241.471,A -85,B 0,C 180,E1 -5887.545,E2 -5887.545} C_VEL
LIN {X 0,Y 502.802,Z 240.856,A -85,B 0,C 180,E1 -5887.952,E2 -5887.952} C_VEL
LIN {X 0,Y 502.759,Z 240.862,A -85,B 0,C 180,E1 -5891.071,E2 -5891.071} C_VEL
LIN {X 0,Y 502.775,Z 240.858,A -85,B 0,C 180,E1 -5894.528,E2 -5894.528} C_VEL
LIN {X 0,Y 502.762,Z 240.856,A -85,B 0,C 180,E1 -5897.856,E2 -5897.856} C_VEL
LIN {X 0,Y 502.773,Z 240.856,A -85,B 0,C 180,E1 -5901.021,E2 -5901.021} C_VEL
LIN {X 0,Y 502.746,Z 240.862,A -85,B 0,C 180,E1 -5904.172,E2 -5904.172} C_VEL
LIN {X 0,Y 502.826,Z 240.848,A -85,B 0,C 180,E1 -5906.993,E2 -5906.993} C_VEL
LIN {X 0,Y 502.808,Z 240.855,A -85,B 0,C 180,E1 -5910.064,E2 -5910.064} C_VEL
LIN {X 0,Y 502.794,Z 240.854,A -85,B 0,C 180,E1 -5913.453,E2 -5913.453} C_VEL
LIN {X 0,Y 502.767,Z 240.861,A -85,B 0,C 180,E1 -5916.084,E2 -5916.084} C_VEL
LIN {X 0,Y 502.776,Z 240.855,A -85,B 0,C 180,E1 -5918.688,E2 -5918.688} C_VEL
LIN {X 0,Y 502.818,Z 240.853,A -85,B 0,C 180,E1 -5921.247,E2 -5921.247} C_VEL
LIN {X 0,Y 502.841,Z 240.847,A -85,B 0,C 180,E1 -5924.599,E2 -5924.599} C_VEL
LIN {X 0,Y 502.868,Z 240.844,A -85,B 0,C 180,E1 -5928.038,E2 -5928.038} C_VEL
LIN {X 0,Y 502.865,Z 240.848,A -85,B 0,C 180,E1 -5931.156,E2 -5931.156} C_VEL
LIN {X 0,Y 502.918,Z 240.839,A -85,B 0,C 180,E1 -5933.58,E2 -5933.58} C_VEL
LIN {X 0,Y 502.89,Z 240.845,A -85,B 0,C 180,E1 -5936.795,E2 -5936.795} C_VEL
LIN {X 0,Y 503.026,Z 240.827,A -85,B 0,C 180,E1 -5939.199,E2 -5939.199} C_VEL
LIN {X 0,Y 502.894,Z 240.84,A -85,B 0,C 180,E1 -5941.601,E2 -5941.601} C_VEL
LIN {X 0,Y 502.893,Z 240.842,A -85,B 0,C 180,E1 -5943.204,E2 -5943.204} C_VEL
LIN {X 0,Y 502.918,Z 240.842,A -85,B 0,C 180,E1 -5946.418,E2 -5946.418} C_VEL
LIN {X 0,Y 502.867,Z 240.846,A -85,B 0,C 180,E1 -5948.842,E2 -5948.842} C_VEL
LIN {X 0,Y 502.851,Z 240.851,A -85,B 0,C 180,E1 -5952.1,E2 -5952.1} C_VEL
LIN {X 0,Y 502.837,Z 240.847,A -85,B 0,C 180,E1 -5955.399,E2 -5955.399} C_VEL
LIN {X 0,Y 502.834,Z 240.851,A -85,B 0,C 180,E1 -5958.122,E2 -5958.122} C_VEL
LIN {X 0,Y 502.816,Z 240.85,A -85,B 0,C 180,E1 -5960.535,E2 -5960.535} C_VEL
LIN {X 0,Y 502.784,Z 240.854,A -85,B 0,C 180,E1 -5963.04,E2 -5963.04} C_VEL
LIN {X 0,Y 502.829,Z 240.853,A -85,B 0,C 180,E1 -5965.675,E2 -5965.675} C_VEL
LIN {X 0,Y 502.83,Z 240.847,A -85,B 0,C 180,E1 -5968.372,E2 -5968.372} C_VEL
LIN {X 0,Y 502.784,Z 240.858,A -85,B 0,C 180,E1 -5971.499,E2 -5971.499} C_VEL
LIN {X 0,Y 502.794,Z 240.851,A -85,B 0,C 180,E1 -5974.444,E2 -5974.444} C_VEL
LIN {X 0,Y 502.771,Z 240.861,A -85,B 0,C 180,E1 -5977.178,E2 -5977.178} C_VEL
LIN {X 0,Y 502.814,Z 240.848,A -85,B 0,C 180,E1 -5980.011,E2 -5980.011} C_VEL
LIN {X 0,Y 502.814,Z 240.848,A -85,B 0,C 180,E1 -5982.202,E2 -5982.202} C_VEL
LIN {X 0,Y 502.787,Z 240.852,A -85,B 0,C 180,E1 -5985.468,E2 -5985.468} C_VEL
LIN {X 0,Y 502.817,Z 240.848,A -85,B 0,C 180,E1 -5987.864,E2 -5987.864} C_VEL
LIN {X 0,Y 502.789,Z 240.854,A -85,B 0,C 180,E1 -5991.024,E2 -5991.024} C_VEL
LIN {X 0,Y 502.769,Z 240.858,A -85,B 0,C 180,E1 -5994.168,E2 -5994.168} C_VEL
LIN {X 0,Y 502.794,Z 240.851,A -85,B 0,C 180,E1 -5997.237,E2 -5997.237} C_VEL
LIN {X 0,Y 502.094,Z 240.942,A -85,B 0,C 180,E1 -5997.906,E2 -5997.906} C_VEL
LIN {X 0,Y 499.229,Z 241.299,A -85,B 0,C 180,E1 -5998.991,E2 -5998.991} C_VEL
LIN {X 0,Y 496.834,Z 241.598,A -85,B 0,C 180,E1 -5999.866,E2 -5999.866} C_VEL
LIN {X 0,Y 495.818,Z 241.725,A -85,B 0,C 180,E1 -6000.542,E2 -6000.542} C_VEL
LIN {X 0,Y 495.74,Z 241.731,A -85,B 0,C 180,E1 -6000.771,E2 -6000.771} C_VEL
LIN {X 0,Y 495.793,Z 241.724,A -85,B 0,C 180,E1 -6003.255,E2 -6003.255} C_VEL
LIN {X 0,Y 495.707,Z 241.738,A -85,B 0,C 180,E1 -6005.723,E2 -6005.723} C_VEL
LIN {X 0,Y 495.674,Z 241.741,A -85,B 0,C 180,E1 -6007.492,E2 -6007.492} C_VEL
LIN {X 0,Y 495.58,Z 242.171,A -85,B 0,C 180,E1 -6008.364,E2 -6008.364} C_VEL
LIN {X 0,Y 495.558,Z 246.065,A -85,B 0,C 180,E1 -6010.963,E2 -6010.963} C_VEL
LIN {X 0,Y 495.5,Z 249.97,A -85,B 0,C 180,E1 -6013.521,E2 -6013.521} C_VEL
LIN {X 0,Y 495.418,Z 253.87,A -85,B 0,C 180,E1 -6016.045,E2 -6016.045} C_VEL
LIN {X 0,Y 495.428,Z 257.766,A -85,B 0,C 180,E1 -6018.545,E2 -6018.545} C_VEL
LIN {X 0,Y 495.321,Z 263.012,A -85,B 0,C 180,E1 -6021.843,E2 -6021.843} C_VEL
LIN {X 0,Y 495.26,Z 266.962,A -85,B 0,C 180,E1 -6024.299,E2 -6024.299} C_VEL
LIN {X 0,Y 495.238,Z 270.948,A -85,B 0,C 180,E1 -6026.746,E2 -6026.746} C_VEL
LIN {X 0,Y 495.092,Z 274.057,A -85,B 0,C 180,E1 -6028.577,E2 -6028.577} C_VEL
LIN {X 0,Y 497.706,Z 287.226,A -85,B 0,C 180,E1 -6029.014,E2 -6029.014} C_VEL
LIN {X 0,Y 497.442,Z 300.392,A -85,B 0,C 180,E1 -6029.545,E2 -6029.545} C_VEL
LIN {X 0,Y 497.105,Z 312.3,A -85,B 0,C 180,E1 -6030.202,E2 -6030.202} C_VEL
LIN {X 0,Y 496.701,Z 323.673,A -85,B 0,C 180,E1 -6031.013,E2 -6031.013} C_VEL
LIN {X 0,Y 496.323,Z 333.938,A -85,B 0,C 180,E1 -6031.927,E2 -6031.927} C_VEL
LIN {X 0,Y 496.017,Z 342.353,A -85,B 0,C 180,E1 -6032.842,E2 -6032.842} C_VEL
LIN {X 0,Y 495.692,Z 350.147,A -85,B 0,C 180,E1 -6033.861,E2 -6033.861} C_VEL
LIN {X 0,Y 495.443,Z 357.771,A -85,B 0,C 180,E1 -6035.086,E2 -6035.086} C_VEL
LIN {X 0,Y 495.237,Z 364.813,A -85,B 0,C 180,E1 -6036.519,E2 -6036.519} C_VEL
LIN {X 0,Y 495.138,Z 369.511,A -85,B 0,C 180,E1 -6037.749,E2 -6037.749} C_VEL
LIN {X 0,Y 495.04,Z 373.116,A -85,B 0,C 180,E1 -6038.984,E2 -6038.984} C_VEL
LIN {X 0,Y 494.97,Z 374.973,A -85,B 0,C 180,E1 -6039.81,E2 -6039.81} C_VEL
LIN {X 0,Y 494.981,Z 376.355,A -85,B 0,C 180,E1 -6040.636,E2 -6040.636} C_VEL
LIN {X 0,Y 495.009,Z 377.46,A -85,B 0,C 180,E1 -6041.588,E2 -6041.588} C_VEL
LIN {X 0,Y 494.908,Z 378.101,A -85,B 0,C 180,E1 -6043.132,E2 -6043.132} C_VEL
LIN {X 0,Y 494.908,Z 377.834,A -85,B 0,C 180,E1 -6043.969,E2 -6043.969} C_VEL
LIN {X 0,Y 494.941,Z 376.872,A -85,B 0,C 180,E1 -6045.083,E2 -6045.083} C_VEL
LIN {X 0,Y 494.95,Z 374.522,A -85,B 0,C 180,E1 -6046.498,E2 -6046.498} C_VEL
LIN {X 0,Y 495.113,Z 370.607,A -85,B 0,C 180,E1 -6048.007,E2 -6048.007} C_VEL
LIN {X 0,Y 495.248,Z 365.24,A -85,B 0,C 180,E1 -6049.48,E2 -6049.48} C_VEL
LIN {X 0,Y 495.422,Z 359.061,A -85,B 0,C 180,E1 -6050.771,E2 -6050.771} C_VEL
LIN {X 0,Y 495.699,Z 351.258,A -85,B 0,C 180,E1 -6052.068,E2 -6052.068} C_VEL
LIN {X 0,Y 496.013,Z 342.655,A -85,B 0,C 180,E1 -6053.217,E2 -6053.217} C_VEL
LIN {X 0,Y 496.368,Z 333.155,A -85,B 0,C 180,E1 -6054.242,E2 -6054.242} C_VEL
LIN {X 0,Y 496.754,Z 321.849,A -85,B 0,C 180,E1 -6055.226,E2 -6055.226} C_VEL
LIN {X 0,Y 497.169,Z 310.713,A -85,B 0,C 180,E1 -6055.989,E2 -6055.989} C_VEL
LIN {X 0,Y 497.53,Z 299.454,A -85,B 0,C 180,E1 -6056.59,E2 -6056.59} C_VEL
LIN {X 0,Y 497.67,Z 287.249,A -85,B 0,C 180,E1 -6057.08,E2 -6057.08} C_VEL
LIN {X 0,Y 495.077,Z 274.004,A -85,B 0,C 180,E1 -6057.538,E2 -6057.538} C_VEL
LIN {X 0,Y 495.128,Z 268.819,A -85,B 0,C 180,E1 -6060.729,E2 -6060.729} C_VEL
LIN {X 0,Y 495.216,Z 264.228,A -85,B 0,C 180,E1 -6063.605,E2 -6063.605} C_VEL
LIN {X 0,Y 495.313,Z 259.577,A -85,B 0,C 180,E1 -6066.578,E2 -6066.578} C_VEL
LIN {X 0,Y 495.402,Z 254.846,A -85,B 0,C 180,E1 -6069.671,E2 -6069.671} C_VEL
LIN {X 0,Y 495.497,Z 250.646,A -85,B 0,C 180,E1 -6072.479,E2 -6072.479} C_VEL
LIN {X 0,Y 495.673,Z 246.749,A -85,B 0,C 180,E1 -6075.147,E2 -6075.147} C_VEL
LIN {X 0,Y 495.677,Z 242.39,A -85,B 0,C 180,E1 -6078.212,E2 -6078.212} C_VEL
LIN {X 0,Y 495.682,Z 241.746,A -85,B 0,C 180,E1 -6078.715,E2 -6078.715} C_VEL
LIN {X 0,Y 495.737,Z 241.738,A -85,B 0,C 180,E1 -6081.409,E2 -6081.409} C_VEL
LIN {X 0,Y 495.745,Z 241.737,A -85,B 0,C 180,E1 -6084.464,E2 -6084.464} C_VEL
LIN {X 0,Y 495.755,Z 241.736,A -85,B 0,C 180,E1 -6087.406,E2 -6087.406} C_VEL
LIN {X 0,Y 495.769,Z 241.734,A -85,B 0,C 180,E1 -6090.255,E2 -6090.255} C_VEL
LIN {X 0,Y 495.81,Z 241.727,A -85,B 0,C 180,E1 -6093.251,E2 -6093.251} C_VEL
LIN {X 0,Y 495.746,Z 241.732,A -85,B 0,C 180,E1 -6095.726,E2 -6095.726} C_VEL
LIN {X 0,Y 495.752,Z 241.732,A -85,B 0,C 180,E1 -6098.373,E2 -6098.373} C_VEL
LIN {X 0,Y 495.771,Z 241.732,A -85,B 0,C 180,E1 -6100.972,E2 -6100.972} C_VEL
LIN {X 0,Y 495.769,Z 241.73,A -85,B 0,C 180,E1 -6103.531,E2 -6103.531} C_VEL
LIN {X 0,Y 495.779,Z 241.727,A -85,B 0,C 180,E1 -6106.056,E2 -6106.056} C_VEL
LIN {X 0,Y 495.84,Z 241.724,A -85,B 0,C 180,E1 -6108.556,E2 -6108.556} C_VEL
LIN {X 0,Y 495.863,Z 241.718,A -85,B 0,C 180,E1 -6111.853,E2 -6111.853} C_VEL
LIN {X 0,Y 495.873,Z 241.719,A -85,B 0,C 180,E1 -6114.307,E2 -6114.307} C_VEL
LIN {X 0,Y 495.984,Z 241.706,A -85,B 0,C 180,E1 -6117.565,E2 -6117.565} C_VEL
LIN {X 0,Y 495.983,Z 241.702,A -85,B 0,C 180,E1 -6120.001,E2 -6120.001} C_VEL
LIN {X 0,Y 495.986,Z 241.703,A -85,B 0,C 180,E1 -6122.437,E2 -6122.437} C_VEL
LIN {X 0,Y 495.879,Z 241.715,A -85,B 0,C 180,E1 -6125.695,E2 -6125.695} C_VEL
LIN {X 0,Y 495.863,Z 241.721,A -85,B 0,C 180,E1 -6128.149,E2 -6128.149} C_VEL
LIN {X 0,Y 495.847,Z 241.72,A -85,B 0,C 180,E1 -6131.446,E2 -6131.446} C_VEL
LIN {X 0,Y 495.78,Z 241.728,A -85,B 0,C 180,E1 -6134.784,E2 -6134.784} C_VEL
LIN {X 0,Y 495.778,Z 241.732,A -85,B 0,C 180,E1 -6137.32,E2 -6137.32} C_VEL
LIN {X 0,Y 495.763,Z 241.734,A -85,B 0,C 180,E1 -6139.892,E2 -6139.892} C_VEL
LIN {X 0,Y 495.755,Z 241.735,A -85,B 0,C 180,E1 -6142.862,E2 -6142.862} C_VEL
LIN {X 0,Y 495.777,Z 241.734,A -85,B 0,C 180,E1 -6146.069,E2 -6146.069} C_VEL
LIN {X 0,Y 495.738,Z 241.737,A -85,B 0,C 180,E1 -6148.818,E2 -6148.818} C_VEL
LIN {X 0,Y 495.752,Z 241.733,A -85,B 0,C 180,E1 -6151.727,E2 -6151.727} C_VEL
LIN {X 0,Y 495.763,Z 241.731,A -85,B 0,C 180,E1 -6154.695,E2 -6154.695} C_VEL
LIN {X 0,Y 495.725,Z 241.735,A -85,B 0,C 180,E1 -6157.563,E2 -6157.563} C_VEL
LIN {X 0,Y 495.763,Z 241.728,A -85,B 0,C 180,E1 -6160.701,E2 -6160.701} C_VEL
LIN {X 0,Y 495.725,Z 241.737,A -85,B 0,C 180,E1 -6164.003,E2 -6164.003} C_VEL
LIN {X 0,Y 495.701,Z 241.744,A -85,B 0,C 180,E1 -6167.116,E2 -6167.116} C_VEL
LIN {X 0,Y 495.749,Z 241.735,A -85,B 0,C 180,E1 -6170.363,E2 -6170.363} C_VEL
LIN {X 0,Y 495.781,Z 241.953,A -85,B 0,C 180,E1 -6171.412,E2 -6171.412} C_VEL
LIN {X 0,Y 496.502,Z 246.61,A -85,B 0,C 180,E1 -6173.789,E2 -6173.789} C_VEL
LIN {X 0,Y 496.593,Z 251.309,A -85,B 0,C 180,E1 -6176.013,E2 -6176.013} C_VEL
LIN {X 0,Y 496.274,Z 257.687,A -85,B 0,C 180,E1 -6178.877,E2 -6178.877} C_VEL
LIN {X 0,Y 496.042,Z 263.648,A -85,B 0,C 180,E1 -6181.454,E2 -6181.454} C_VEL
LIN {X 0,Y 495.773,Z 271.76,A -85,B 0,C 180,E1 -6184.833,E2 -6184.833} C_VEL
LIN {X 0,Y 495.591,Z 279.458,A -85,B 0,C 180,E1 -6187.927,E2 -6187.927} C_VEL
LIN {X 0,Y 495.405,Z 287.202,A -85,B 0,C 180,E1 -6190.957,E2 -6190.957} C_VEL
LIN {X 0,Y 495.265,Z 294.981,A -85,B 0,C 180,E1 -6193.936,E2 -6193.936} C_VEL
LIN {X 0,Y 495.221,Z 299.097,A -85,B 0,C 180,E1 -6195.489,E2 -6195.489} C_VEL
LIN {X 0,Y 497.427,Z 313.228,A -85,B 0,C 180,E1 -6195.92,E2 -6195.92} C_VEL
LIN {X 0,Y 497.578,Z 318.423,A -85,B 0,C 180,E1 -6196.107,E2 -6196.107} C_VEL
LIN {X 0,Y 497.221,Z 330.077,A -85,B 0,C 180,E1 -6196.618,E2 -6196.618} C_VEL
LIN {X 0,Y 496.821,Z 342.298,A -85,B 0,C 180,E1 -6197.328,E2 -6197.328} C_VEL
LIN {X 0,Y 496.49,Z 353.397,A -85,B 0,C 180,E1 -6198.156,E2 -6198.156} C_VEL
LIN {X 0,Y 496.097,Z 364.299,A -85,B 0,C 180,E1 -6199.181,E2 -6199.181} C_VEL
LIN {X 0,Y 495.743,Z 373.158,A -85,B 0,C 180,E1 -6200.205,E2 -6200.205} C_VEL
LIN {X 0,Y 495.477,Z 381.8,A -85,B 0,C 180,E1 -6201.435,E2 -6201.435} C_VEL
LIN {X 0,Y 495.274,Z 388.707,A -85,B 0,C 180,E1 -6202.663,E2 -6202.663} C_VEL
LIN {X 0,Y 495.12,Z 394.792,A -85,B 0,C 180,E1 -6204.027,E2 -6204.027} C_VEL
LIN {X 0,Y 495.037,Z 398.585,A -85,B 0,C 180,E1 -6205.114,E2 -6205.114} C_VEL
LIN {X 0,Y 495.032,Z 400.884,A -85,B 0,C 180,E1 -6205.93,E2 -6205.93} C_VEL
LIN {X 0,Y 495.042,Z 402.749,A -85,B 0,C 180,E1 -6206.745,E2 -6206.745} C_VEL
LIN {X 0,Y 494.999,Z 404.146,A -85,B 0,C 180,E1 -6207.559,E2 -6207.559} C_VEL
LIN {X 0,Y 494.963,Z 405.143,A -85,B 0,C 180,E1 -6208.373,E2 -6208.373} C_VEL
LIN {X 0,Y 494.898,Z 405.969,A -85,B 0,C 180,E1 -6210,E2 -6210} C_VEL
LIN {X 0,Y 494.963,Z 405.15,A -85,B 0,C 180,E1 -6211.627,E2 -6211.627} C_VEL
LIN {X 0,Y 494.999,Z 404.157,A -85,B 0,C 180,E1 -6212.441,E2 -6212.441} C_VEL
LIN {X 0,Y 495.042,Z 402.764,A -85,B 0,C 180,E1 -6213.255,E2 -6213.255} C_VEL
LIN {X 0,Y 495.009,Z 399.828,A -85,B 0,C 180,E1 -6214.479,E2 -6214.479} C_VEL
LIN {X 0,Y 495.129,Z 395.857,A -85,B 0,C 180,E1 -6215.702,E2 -6215.702} C_VEL
LIN {X 0,Y 495.258,Z 389.747,A -85,B 0,C 180,E1 -6217.133,E2 -6217.133} C_VEL
LIN {X 0,Y 495.431,Z 383.069,A -85,B 0,C 180,E1 -6218.36,E2 -6218.36} C_VEL
LIN {X 0,Y 495.706,Z 374.784,A -85,B 0,C 180,E1 -6219.589,E2 -6219.589} C_VEL
LIN {X 0,Y 495.999,Z 366.292,A -85,B 0,C 180,E1 -6220.614,E2 -6220.614} C_VEL
LIN {X 0,Y 496.404,Z 355.8,A -85,B 0,C 180,E1 -6221.639,E2 -6221.639} C_VEL
LIN {X 0,Y 496.749,Z 344.581,A -85,B 0,C 180,E1 -6222.521,E2 -6222.521} C_VEL
LIN {X 0,Y 497.151,Z 334.046,A -85,B 0,C 180,E1 -6223.176,E2 -6223.176} C_VEL
LIN {X 0,Y 497.502,Z 322.373,A -85,B 0,C 180,E1 -6223.739,E2 -6223.739} C_VEL
LIN {X 0,Y 497.471,Z 313.657,A -85,B 0,C 180,E1 -6224.066,E2 -6224.066} C_VEL
LIN {X 0,Y 495.459,Z 300.819,A -85,B 0,C 180,E1 -6224.465,E2 -6224.465} C_VEL
LIN {X 0,Y 495.221,Z 299.157,A -85,B 0,C 180,E1 -6224.511,E2 -6224.511} C_VEL
LIN {X 0,Y 495.336,Z 291.708,A -85,B 0,C 180,E1 -6227.334,E2 -6227.334} C_VEL
LIN {X 0,Y 495.46,Z 285.017,A -85,B 0,C 180,E1 -6229.903,E2 -6229.903} C_VEL
LIN {X 0,Y 495.601,Z 277.553,A -85,B 0,C 180,E1 -6232.816,E2 -6232.816} C_VEL
LIN {X 0,Y 495.836,Z 269.394,A -85,B 0,C 180,E1 -6236.065,E2 -6236.065} C_VEL
LIN {X 0,Y 496.042,Z 261.59,A -85,B 0,C 180,E1 -6239.261,E2 -6239.261} C_VEL
LIN {X 0,Y 496.271,Z 255.498,A -85,B 0,C 180,E1 -6241.82,E2 -6241.82} C_VEL
LIN {X 0,Y 496.473,Z 248.611,A -85,B 0,C 180,E1 -6244.81,E2 -6244.81} C_VEL
LIN {X 0,Y 496.127,Z 243.845,A -85,B 0,C 180,E1 -6246.985,E2 -6246.985} C_VEL
LIN {X 0,Y 495.766,Z 241.733,A -85,B 0,C 180,E1 -6248.071,E2 -6248.071} C_VEL
LIN {X 0,Y 495.724,Z 241.738,A -85,B 0,C 180,E1 -6250.703,E2 -6250.703} C_VEL
LIN {X 0,Y 495.71,Z 241.734,A -85,B 0,C 180,E1 -6254.002,E2 -6254.002} C_VEL
LIN {X 0,Y 495.685,Z 241.739,A -85,B 0,C 180,E1 -6257.112,E2 -6257.112} C_VEL
LIN {X 0,Y 495.734,Z 241.735,A -85,B 0,C 180,E1 -6260.359,E2 -6260.359} C_VEL
LIN {X 0,Y 495.682,Z 241.738,A -85,B 0,C 180,E1 -6263.451,E2 -6263.451} C_VEL
LIN {X 0,Y 495.748,Z 241.735,A -85,B 0,C 180,E1 -6266.434,E2 -6266.434} C_VEL
LIN {X 0,Y 495.744,Z 241.731,A -85,B 0,C 180,E1 -6269.311,E2 -6269.311} C_VEL
LIN {X 0,Y 495.72,Z 241.739,A -85,B 0,C 180,E1 -6272.104,E2 -6272.104} C_VEL
LIN {X 0,Y 495.728,Z 241.733,A -85,B 0,C 180,E1 -6275.137,E2 -6275.137} C_VEL
LIN {X 0,Y 495.741,Z 241.734,A -85,B 0,C 180,E1 -6277.494,E2 -6277.494} C_VEL
LIN {X 0,Y 495.763,Z 241.731,A -85,B 0,C 180,E1 -6280.108,E2 -6280.108} C_VEL
LIN {X 0,Y 495.757,Z 241.729,A -85,B 0,C 180,E1 -6282.68,E2 -6282.68} C_VEL
LIN {X 0,Y 495.782,Z 241.729,A -85,B 0,C 180,E1 -6285.216,E2 -6285.216} C_VEL
LIN {X 0,Y 495.843,Z 241.719,A -85,B 0,C 180,E1 -6288.554,E2 -6288.554} C_VEL
LIN {X 0,Y 495.864,Z 241.717,A -85,B 0,C 180,E1 -6291.851,E2 -6291.851} C_VEL
LIN {X 0,Y 495.886,Z 241.714,A -85,B 0,C 180,E1 -6294.305,E2 -6294.305} C_VEL
LIN {X 0,Y 495.983,Z 241.702,A -85,B 0,C 180,E1 -6297.563,E2 -6297.563} C_VEL
LIN {X 0,Y 495.986,Z 241.701,A -85,B 0,C 180,E1 -6299.999,E2 -6299.999} C_VEL
LIN {X 0,Y 495.983,Z 241.706,A -85,B 0,C 180,E1 -6302.435,E2 -6302.435} C_VEL
LIN {X 0,Y 495.894,Z 241.712,A -85,B 0,C 180,E1 -6305.692,E2 -6305.692} C_VEL
LIN {X 0,Y 495.863,Z 241.72,A -85,B 0,C 180,E1 -6308.147,E2 -6308.147} C_VEL
LIN {X 0,Y 495.844,Z 241.718,A -85,B 0,C 180,E1 -6311.444,E2 -6311.444} C_VEL
LIN {X 0,Y 495.779,Z 241.727,A -85,B 0,C 180,E1 -6314.782,E2 -6314.782} C_VEL
LIN {X 0,Y 495.776,Z 241.727,A -85,B 0,C 180,E1 -6317.318,E2 -6317.318} C_VEL
LIN {X 0,Y 495.767,Z 241.733,A -85,B 0,C 180,E1 -6319.889,E2 -6319.889} C_VEL
LIN {X 0,Y 495.753,Z 241.729,A -85,B 0,C 180,E1 -6322.862,E2 -6322.862} C_VEL
LIN {X 0,Y 495.787,Z 241.727,A -85,B 0,C 180,E1 -6326.067,E2 -6326.067} C_VEL
LIN {X 0,Y 495.768,Z 241.727,A -85,B 0,C 180,E1 -6328.814,E2 -6328.814} C_VEL
LIN {X 0,Y 495.747,Z 241.732,A -85,B 0,C 180,E1 -6331.726,E2 -6331.726} C_VEL
LIN {X 0,Y 495.764,Z 241.728,A -85,B 0,C 180,E1 -6334.695,E2 -6334.695} C_VEL
LIN {X 0,Y 495.722,Z 241.735,A -85,B 0,C 180,E1 -6337.561,E2 -6337.561} C_VEL
LIN {X 0,Y 495.781,Z 241.724,A -85,B 0,C 180,E1 -6340.052,E2 -6340.052} C_VEL
LIN {X 0,Y 495.751,Z 241.735,A -85,B 0,C 180,E1 -6342.879,E2 -6342.879} C_VEL
LIN {X 0,Y 495.723,Z 241.731,A -85,B 0,C 180,E1 -6345.999,E2 -6345.999} C_VEL
LIN {X 0,Y 495.751,Z 241.736,A -85,B 0,C 180,E1 -6348.706,E2 -6348.706} C_VEL
LIN {X 0,Y 495.738,Z 241.73,A -85,B 0,C 180,E1 -6351.408,E2 -6351.408} C_VEL
LIN {X 0,Y 495.742,Z 241.737,A -85,B 0,C 180,E1 -6354.463,E2 -6354.463} C_VEL
LIN {X 0,Y 495.755,Z 241.728,A -85,B 0,C 180,E1 -6357.406,E2 -6357.406} C_VEL
LIN {X 0,Y 495.754,Z 241.735,A -85,B 0,C 180,E1 -6360.254,E2 -6360.254} C_VEL
LIN {X 0,Y 495.74,Z 241.731,A -85,B 0,C 180,E1 -6360.771,E2 -6360.771} C_VEL
LIN {X 0,Y 495.081,Z 241.814,A -85,B 0,C 180,E1 -6361.45,E2 -6361.45} C_VEL
LIN {X 0,Y 492.216,Z 242.172,A -85,B 0,C 180,E1 -6362.552,E2 -6362.552} C_VEL
LIN {X 0,Y 489.798,Z 242.472,A -85,B 0,C 180,E1 -6363.44,E2 -6363.44} C_VEL
LIN {X 0,Y 488.774,Z 242.605,A -85,B 0,C 180,E1 -6364.126,E2 -6364.126} C_VEL
LIN {X 0,Y 488.7,Z 242.61,A -85,B 0,C 180,E1 -6364.358,E2 -6364.358} C_VEL
LIN {X 0,Y 488.668,Z 242.612,A -85,B 0,C 180,E1 -6367.151,E2 -6367.151} C_VEL
LIN {X 0,Y 488.53,Z 242.635,A -85,B 0,C 180,E1 -6368.036,E2 -6368.036} C_VEL
LIN {X 0,Y 488.514,Z 246.443,A -85,B 0,C 180,E1 -6370.678,E2 -6370.678} C_VEL
LIN {X 0,Y 488.434,Z 250.358,A -85,B 0,C 180,E1 -6373.275,E2 -6373.275} C_VEL
LIN {X 0,Y 488.365,Z 254.274,A -85,B 0,C 180,E1 -6375.839,E2 -6375.839} C_VEL
LIN {X 0,Y 488.393,Z 258.195,A -85,B 0,C 180,E1 -6378.378,E2 -6378.378} C_VEL
LIN {X 0,Y 488.267,Z 263.455,A -85,B 0,C 180,E1 -6381.724,E2 -6381.724} C_VEL
LIN {X 0,Y 488.203,Z 267.424,A -85,B 0,C 180,E1 -6384.217,E2 -6384.217} C_VEL
LIN {X 0,Y 488.184,Z 271.416,A -85,B 0,C 180,E1 -6386.699,E2 -6386.699} C_VEL
LIN {X 0,Y 487.966,Z 274.111,A -85,B 0,C 180,E1 -6388.349,E2 -6388.349} C_VEL
LIN {X 0,Y 490.831,Z 288.288,A -85,B 0,C 180,E1 -6388.846,E2 -6388.846} C_VEL
LIN {X 0,Y 490.519,Z 301.237,A -85,B 0,C 180,E1 -6389.384,E2 -6389.384} C_VEL
LIN {X 0,Y 490.141,Z 313.745,A -85,B 0,C 180,E1 -6390.103,E2 -6390.103} C_VEL
LIN {X 0,Y 489.734,Z 324.889,A -85,B 0,C 180,E1 -6390.925,E2 -6390.925} C_VEL
LIN {X 0,Y 489.311,Z 334.977,A -85,B 0,C 180,E1 -6391.852,E2 -6391.852} C_VEL
LIN {X 0,Y 488.922,Z 344.068,A -85,B 0,C 180,E1 -6392.884,E2 -6392.884} C_VEL
LIN {X 0,Y 488.578,Z 352.932,A -85,B 0,C 180,E1 -6394.124,E2 -6394.124} C_VEL
LIN {X 0,Y 488.279,Z 360.099,A -85,B 0,C 180,E1 -6395.368,E2 -6395.368} C_VEL
LIN {X 0,Y 488.167,Z 365.818,A -85,B 0,C 180,E1 -6396.613,E2 -6396.613} C_VEL
LIN {X 0,Y 488.065,Z 370.338,A -85,B 0,C 180,E1 -6397.862,E2 -6397.862} C_VEL
LIN {X 0,Y 487.946,Z 373.789,A -85,B 0,C 180,E1 -6399.116,E2 -6399.116} C_VEL
LIN {X 0,Y 487.895,Z 375.506,A -85,B 0,C 180,E1 -6399.954,E2 -6399.954} C_VEL
LIN {X 0,Y 487.889,Z 376.814,A -85,B 0,C 180,E1 -6400.793,E2 -6400.793} C_VEL
LIN {X 0,Y 487.914,Z 377.724,A -85,B 0,C 180,E1 -6401.634,E2 -6401.634} C_VEL
LIN {X 0,Y 487.832,Z 378.207,A -85,B 0,C 180,E1 -6402.48,E2 -6402.48} C_VEL
LIN {X 0,Y 487.803,Z 378.264,A -85,B 0,C 180,E1 -6403.327,E2 -6403.327} C_VEL
LIN {X 0,Y 487.831,Z 377.922,A -85,B 0,C 180,E1 -6404.176,E2 -6404.176} C_VEL
LIN {X 0,Y 487.86,Z 376.995,A -85,B 0,C 180,E1 -6405.169,E2 -6405.169} C_VEL
LIN {X 0,Y 487.883,Z 374.302,A -85,B 0,C 180,E1 -6406.744,E2 -6406.744} C_VEL
LIN {X 0,Y 488.048,Z 370.674,A -85,B 0,C 180,E1 -6408.123,E2 -6408.123} C_VEL
LIN {X 0,Y 488.168,Z 366.391,A -85,B 0,C 180,E1 -6409.336,E2 -6409.336} C_VEL
LIN {X 0,Y 488.336,Z 360.235,A -85,B 0,C 180,E1 -6410.701,E2 -6410.701} C_VEL
LIN {X 0,Y 488.612,Z 353.011,A -85,B 0,C 180,E1 -6411.96,E2 -6411.96} C_VEL
LIN {X 0,Y 488.976,Z 344.027,A -85,B 0,C 180,E1 -6413.219,E2 -6413.219} C_VEL
LIN {X 0,Y 489.356,Z 334.702,A -85,B 0,C 180,E1 -6414.274,E2 -6414.274} C_VEL
LIN {X 0,Y 489.751,Z 324.465,A -85,B 0,C 180,E1 -6415.208,E2 -6415.208} C_VEL
LIN {X 0,Y 490.146,Z 312.99,A -85,B 0,C 180,E1 -6416.047,E2 -6416.047} C_VEL
LIN {X 0,Y 490.533,Z 302.263,A -85,B 0,C 180,E1 -6416.662,E2 -6416.662} C_VEL
LIN {X 0,Y 490.88,Z 289.776,A -85,B 0,C 180,E1 -6417.201,E2 -6417.201} C_VEL
LIN {X 0,Y 489.284,Z 280.29,A -85,B 0,C 180,E1 -6417.554,E2 -6417.554} C_VEL
LIN {X 0,Y 488.01,Z 274.203,A -85,B 0,C 180,E1 -6417.758,E2 -6417.758} C_VEL
LIN {X 0,Y 488.05,Z 268.655,A -85,B 0,C 180,E1 -6421.225,E2 -6421.225} C_VEL
LIN {X 0,Y 488.163,Z 264.044,A -85,B 0,C 180,E1 -6424.157,E2 -6424.157} C_VEL
LIN {X 0,Y 488.274,Z 259.372,A -85,B 0,C 180,E1 -6427.194,E2 -6427.194} C_VEL
LIN {X 0,Y 488.347,Z 254.725,A -85,B 0,C 180,E1 -6430.295,E2 -6430.295} C_VEL
LIN {X 0,Y 488.48,Z 251.034,A -85,B 0,C 180,E1 -6432.799,E2 -6432.799} C_VEL
LIN {X 0,Y 488.642,Z 247.58,A -85,B 0,C 180,E1 -6435.192,E2 -6435.192} C_VEL
LIN {X 0,Y 488.681,Z 244.378,A -85,B 0,C 180,E1 -6437.475,E2 -6437.475} C_VEL
LIN {X 0,Y 488.64,Z 242.869,A -85,B 0,C 180,E1 -6438.579,E2 -6438.579} C_VEL
LIN {X 0,Y 488.69,Z 242.617,A -85,B 0,C 180,E1 -6440.948,E2 -6440.948} C_VEL
LIN {X 0,Y 488.673,Z 242.615,A -85,B 0,C 180,E1 -6443.869,E2 -6443.869} C_VEL
LIN {X 0,Y 488.725,Z 242.61,A -85,B 0,C 180,E1 -6446.878,E2 -6446.878} C_VEL
LIN {X 0,Y 488.721,Z 242.608,A -85,B 0,C 180,E1 -6449.782,E2 -6449.782} C_VEL
LIN {X 0,Y 488.779,Z 242.602,A -85,B 0,C 180,E1 -6453.057,E2 -6453.057} C_VEL
LIN {X 0,Y 488.692,Z 242.615,A -85,B 0,C 180,E1 -6456.256,E2 -6456.256} C_VEL
LIN {X 0,Y 488.735,Z 242.608,A -85,B 0,C 180,E1 -6459.176,E2 -6459.176} C_VEL
LIN {X 0,Y 488.723,Z 242.609,A -85,B 0,C 180,E1 -6462.424,E2 -6462.424} C_VEL
LIN {X 0,Y 488.749,Z 242.604,A -85,B 0,C 180,E1 -6465,E2 -6465} C_VEL
LIN {X 0,Y 488.794,Z 242.602,A -85,B 0,C 180,E1 -6468.388,E2 -6468.388} C_VEL
LIN {X 0,Y 488.808,Z 242.598,A -85,B 0,C 180,E1 -6471.735,E2 -6471.735} C_VEL
LIN {X 0,Y 488.831,Z 242.595,A -85,B 0,C 180,E1 -6474.225,E2 -6474.225} C_VEL
LIN {X 0,Y 488.952,Z 242.582,A -85,B 0,C 180,E1 -6477.53,E2 -6477.53} C_VEL
LIN {X 0,Y 488.955,Z 242.578,A -85,B 0,C 180,E1 -6480.001,E2 -6480.001} C_VEL
LIN {X 0,Y 488.954,Z 242.579,A -85,B 0,C 180,E1 -6482.472,E2 -6482.472} C_VEL
LIN {X 0,Y 488.838,Z 242.592,A -85,B 0,C 180,E1 -6485.777,E2 -6485.777} C_VEL
LIN {X 0,Y 488.808,Z 242.599,A -85,B 0,C 180,E1 -6488.267,E2 -6488.267} C_VEL
LIN {X 0,Y 488.8,Z 242.597,A -85,B 0,C 180,E1 -6491.613,E2 -6491.613} C_VEL
LIN {X 0,Y 488.753,Z 242.604,A -85,B 0,C 180,E1 -6495.002,E2 -6495.002} C_VEL
LIN {X 0,Y 488.748,Z 242.608,A -85,B 0,C 180,E1 -6498.443,E2 -6498.443} C_VEL
LIN {X 0,Y 488.699,Z 242.612,A -85,B 0,C 180,E1 -6501.072,E2 -6501.072} C_VEL
LIN {X 0,Y 488.686,Z 242.614,A -85,B 0,C 180,E1 -6503.747,E2 -6503.747} C_VEL
LIN {X 0,Y 488.723,Z 242.611,A -85,B 0,C 180,E1 -6506.475,E2 -6506.475} C_VEL
LIN {X 0,Y 488.704,Z 242.615,A -85,B 0,C 180,E1 -6509.272,E2 -6509.272} C_VEL
LIN {X 0,Y 488.699,Z 242.615,A -85,B 0,C 180,E1 -6512.148,E2 -6512.148} C_VEL
LIN {X 0,Y 488.712,Z 242.612,A -85,B 0,C 180,E1 -6515.116,E2 -6515.116} C_VEL
LIN {X 0,Y 488.676,Z 242.617,A -85,B 0,C 180,E1 -6518.201,E2 -6518.201} C_VEL
LIN {X 0,Y 488.715,Z 242.606,A -85,B 0,C 180,E1 -6520.346,E2 -6520.346} C_VEL
LIN {X 0,Y 488.682,Z 242.613,A -85,B 0,C 180,E1 -6523.656,E2 -6523.656} C_VEL
LIN {X 0,Y 488.672,Z 242.617,A -85,B 0,C 180,E1 -6526.345,E2 -6526.345} C_VEL
LIN {X 0,Y 488.702,Z 242.613,A -85,B 0,C 180,E1 -6529.675,E2 -6529.675} C_VEL
LIN {X 0,Y 488.747,Z 242.704,A -85,B 0,C 180,E1 -6531.094,E2 -6531.094} C_VEL
LIN {X 0,Y 489.482,Z 247.367,A -85,B 0,C 180,E1 -6533.52,E2 -6533.52} C_VEL
LIN {X 0,Y 489.612,Z 251.317,A -85,B 0,C 180,E1 -6535.46,E2 -6535.46} C_VEL
LIN {X 0,Y 489.323,Z 257.697,A -85,B 0,C 180,E1 -6538.394,E2 -6538.394} C_VEL
LIN {X 0,Y 489.041,Z 264.149,A -85,B 0,C 180,E1 -6541.239,E2 -6541.239} C_VEL
LIN {X 0,Y 488.779,Z 271.694,A -85,B 0,C 180,E1 -6544.447,E2 -6544.447} C_VEL
LIN {X 0,Y 488.546,Z 279.355,A -85,B 0,C 180,E1 -6547.592,E2 -6547.592} C_VEL
LIN {X 0,Y 488.376,Z 285.965,A -85,B 0,C 180,E1 -6550.235,E2 -6550.235} C_VEL
LIN {X 0,Y 488.248,Z 293.707,A -85,B 0,C 180,E1 -6553.269,E2 -6553.269} C_VEL
LIN {X 0,Y 488.124,Z 298.906,A -85,B 0,C 180,E1 -6555.273,E2 -6555.273} C_VEL
LIN {X 0,Y 490.222,Z 312.337,A -85,B 0,C 180,E1 -6555.682,E2 -6555.682} C_VEL
LIN {X 0,Y 490.706,Z 316.902,A -85,B 0,C 180,E1 -6555.856,E2 -6555.856} C_VEL
LIN {X 0,Y 490.364,Z 328.91,A -85,B 0,C 180,E1 -6556.374,E2 -6556.374} C_VEL
LIN {X 0,Y 489.939,Z 341.098,A -85,B 0,C 180,E1 -6557.08,E2 -6557.08} C_VEL
LIN {X 0,Y 489.533,Z 351.935,A -85,B 0,C 180,E1 -6557.88,E2 -6557.88} C_VEL
LIN {X 0,Y 489.209,Z 362.139,A -85,B 0,C 180,E1 -6558.817,E2 -6558.817} C_VEL
LIN {X 0,Y 488.759,Z 371.317,A -85,B 0,C 180,E1 -6559.855,E2 -6559.855} C_VEL
LIN {X 0,Y 488.465,Z 380.268,A -85,B 0,C 180,E1 -6561.103,E2 -6561.103} C_VEL
LIN {X 0,Y 488.228,Z 387.474,A -85,B 0,C 180,E1 -6562.348,E2 -6562.348} C_VEL
LIN {X 0,Y 488.076,Z 392.827,A -85,B 0,C 180,E1 -6563.497,E2 -6563.497} C_VEL
LIN {X 0,Y 488.02,Z 397.069,A -85,B 0,C 180,E1 -6564.629,E2 -6564.629} C_VEL
LIN {X 0,Y 487.928,Z 400.681,A -85,B 0,C 180,E1 -6565.87,E2 -6565.87} C_VEL
LIN {X 0,Y 487.965,Z 402.548,A -85,B 0,C 180,E1 -6566.697,E2 -6566.697} C_VEL
LIN {X 0,Y 487.891,Z 404.943,A -85,B 0,C 180,E1 -6568.349,E2 -6568.349} C_VEL
LIN {X 0,Y 487.819,Z 405.77,A -85,B 0,C 180,E1 -6570,E2 -6570} C_VEL
LIN {X 0,Y 487.891,Z 404.952,A -85,B 0,C 180,E1 -6571.651,E2 -6571.651} C_VEL
LIN {X 0,Y 487.965,Z 402.565,A -85,B 0,C 180,E1 -6573.303,E2 -6573.303} C_VEL
LIN {X 0,Y 487.921,Z 399.629,A -85,B 0,C 180,E1 -6574.544,E2 -6574.544} C_VEL
LIN {X 0,Y 488.027,Z 395.657,A -85,B 0,C 180,E1 -6575.785,E2 -6575.785} C_VEL
LIN {X 0,Y 488.185,Z 389.546,A -85,B 0,C 180,E1 -6577.236,E2 -6577.236} C_VEL
LIN {X 0,Y 488.366,Z 382.868,A -85,B 0,C 180,E1 -6578.482,E2 -6578.482} C_VEL
LIN {X 0,Y 488.674,Z 374.583,A -85,B 0,C 180,E1 -6579.729,E2 -6579.729} C_VEL
LIN {X 0,Y 489.002,Z 366.089,A -85,B 0,C 180,E1 -6580.768,E2 -6580.768} C_VEL
LIN {X 0,Y 489.426,Z 355.592,A -85,B 0,C 180,E1 -6581.807,E2 -6581.807} C_VEL
LIN {X 0,Y 489.8,Z 344.332,A -85,B 0,C 180,E1 -6582.704,E2 -6582.704} C_VEL
LIN {X 0,Y 490.214,Z 333.822,A -85,B 0,C 180,E1 -6583.366,E2 -6583.366} C_VEL
LIN {X 0,Y 490.605,Z 322.131,A -85,B 0,C 180,E1 -6583.936,E2 -6583.936} C_VEL
LIN {X 0,Y 490.559,Z 314.545,A -85,B 0,C 180,E1 -6584.228,E2 -6584.228} C_VEL
LIN {X 0,Y 488.535,Z 301.555,A -85,B 0,C 180,E1 -6584.65,E2 -6584.65} C_VEL
LIN {X 0,Y 488.137,Z 298.959,A -85,B 0,C 180,E1 -6584.726,E2 -6584.726} C_VEL
LIN {X 0,Y 488.262,Z 291.521,A -85,B 0,C 180,E1 -6587.594,E2 -6587.594} C_VEL
LIN {X 0,Y 488.453,Z 283.49,A -85,B 0,C 180,E1 -6590.732,E2 -6590.732} C_VEL
LIN {X 0,Y 488.604,Z 275.911,A -85,B 0,C 180,E1 -6593.749,E2 -6593.749} C_VEL
LIN {X 0,Y 488.832,Z 268.045,A -85,B 0,C 180,E1 -6596.952,E2 -6596.952} C_VEL
LIN {X 0,Y 489.065,Z 260.304,A -85,B 0,C 180,E1 -6600.195,E2 -6600.195} C_VEL
LIN {X 0,Y 489.312,Z 253.621,A -85,B 0,C 180,E1 -6603.078,E2 -6603.078} C_VEL
LIN {X 0,Y 489.458,Z 248.062,A -85,B 0,C 180,E1 -6605.557,E2 -6605.557} C_VEL
LIN {X 0,Y 488.804,Z 243.034,A -85,B 0,C 180,E1 -6607.931,E2 -6607.931} C_VEL
LIN {X 0,Y 488.735,Z 242.609,A -85,B 0,C 180,E1 -6608.194,E2 -6608.194} C_VEL
LIN {X 0,Y 488.658,Z 242.615,A -85,B 0,C 180,E1 -6611.42,E2 -6611.42} C_VEL
LIN {X 0,Y 488.692,Z 242.615,A -85,B 0,C 180,E1 -6614.802,E2 -6614.802} C_VEL
LIN {X 0,Y 488.644,Z 242.614,A -85,B 0,C 180,E1 -6617.468,E2 -6617.468} C_VEL
LIN {X 0,Y 488.7,Z 242.607,A -85,B 0,C 180,E1 -6619.672,E2 -6619.672} C_VEL
LIN {X 0,Y 488.642,Z 242.617,A -85,B 0,C 180,E1 -6622.837,E2 -6622.837} C_VEL
LIN {X 0,Y 488.718,Z 242.608,A -85,B 0,C 180,E1 -6625.885,E2 -6625.885} C_VEL
LIN {X 0,Y 488.685,Z 242.611,A -85,B 0,C 180,E1 -6628.819,E2 -6628.819} C_VEL
LIN {X 0,Y 488.693,Z 242.611,A -85,B 0,C 180,E1 -6631.667,E2 -6631.667} C_VEL
LIN {X 0,Y 488.695,Z 242.611,A -85,B 0,C 180,E1 -6634.441,E2 -6634.441} C_VEL
LIN {X 0,Y 488.715,Z 242.608,A -85,B 0,C 180,E1 -6637.152,E2 -6637.152} C_VEL
LIN {X 0,Y 488.718,Z 242.611,A -85,B 0,C 180,E1 -6639.809,E2 -6639.809} C_VEL
LIN {X 0,Y 488.707,Z 242.608,A -85,B 0,C 180,E1 -6642.422,E2 -6642.422} C_VEL
LIN {X 0,Y 488.754,Z 242.604,A -85,B 0,C 180,E1 -6644.999,E2 -6644.999} C_VEL
LIN {X 0,Y 488.797,Z 242.597,A -85,B 0,C 180,E1 -6648.386,E2 -6648.386} C_VEL
LIN {X 0,Y 488.809,Z 242.597,A -85,B 0,C 180,E1 -6651.733,E2 -6651.733} C_VEL
LIN {X 0,Y 488.845,Z 242.591,A -85,B 0,C 180,E1 -6654.223,E2 -6654.223} C_VEL
LIN {X 0,Y 488.951,Z 242.579,A -85,B 0,C 180,E1 -6657.528,E2 -6657.528} C_VEL
LIN {X 0,Y 488.958,Z 242.577,A -85,B 0,C 180,E1 -6659.999,E2 -6659.999} C_VEL
LIN {X 0,Y 488.951,Z 242.581,A -85,B 0,C 180,E1 -6662.47,E2 -6662.47} C_VEL
LIN {X 0,Y 488.852,Z 242.59,A -85,B 0,C 180,E1 -6665.775,E2 -6665.775} C_VEL
LIN {X 0,Y 488.808,Z 242.599,A -85,B 0,C 180,E1 -6668.265,E2 -6668.265} C_VEL
LIN {X 0,Y 488.797,Z 242.597,A -85,B 0,C 180,E1 -6671.612,E2 -6671.612} C_VEL
LIN {X 0,Y 488.75,Z 242.602,A -85,B 0,C 180,E1 -6675,E2 -6675} C_VEL
LIN {X 0,Y 488.743,Z 242.605,A -85,B 0,C 180,E1 -6678.441,E2 -6678.441} C_VEL
LIN {X 0,Y 488.695,Z 242.609,A -85,B 0,C 180,E1 -6681.07,E2 -6681.07} C_VEL
LIN {X 0,Y 488.682,Z 242.615,A -85,B 0,C 180,E1 -6683.745,E2 -6683.745} C_VEL
LIN {X 0,Y 488.786,Z 242.598,A -85,B 0,C 180,E1 -6686.945,E2 -6686.945} C_VEL
LIN {X 0,Y 488.706,Z 242.607,A -85,B 0,C 180,E1 -6690.364,E2 -6690.364} C_VEL
LIN {X 0,Y 488.723,Z 242.609,A -85,B 0,C 180,E1 -6693.484,E2 -6693.484} C_VEL
LIN {X 0,Y 488.678,Z 242.61,A -85,B 0,C 180,E1 -6696.355,E2 -6696.355} C_VEL
LIN {X 0,Y 488.736,Z 242.607,A -85,B 0,C 180,E1 -6699.249,E2 -6699.249} C_VEL
LIN {X 0,Y 488.721,Z 242.606,A -85,B 0,C 180,E1 -6702.521,E2 -6702.521} C_VEL
LIN {X 0,Y 488.699,Z 242.61,A -85,B 0,C 180,E1 -6705.198,E2 -6705.198} C_VEL
LIN {X 0,Y 488.711,Z 242.609,A -85,B 0,C 180,E1 -6708.398,E2 -6708.398} C_VEL
LIN {X 0,Y 488.691,Z 242.611,A -85,B 0,C 180,E1 -6710.947,E2 -6710.947} C_VEL
LIN {X 0,Y 488.67,Z 242.612,A -85,B 0,C 180,E1 -6713.868,E2 -6713.868} C_VEL
LIN {X 0,Y 488.726,Z 242.606,A -85,B 0,C 180,E1 -6716.877,E2 -6716.877} C_VEL
LIN {X 0,Y 488.711,Z 242.608,A -85,B 0,C 180,E1 -6719.781,E2 -6719.781} C_VEL
LIN {X 0,Y 488.719,Z 242.607,A -85,B 0,C 180,E1 -6722.602,E2 -6722.602} C_VEL
LIN {X 0,Y 488.7,Z 242.61,A -85,B 0,C 180,E1 -6724.358,E2 -6724.358} C_VEL
LIN {X 0,Y 488.046,Z 242.711,A -85,B 0,C 180,E1 -6725.047,E2 -6725.047} C_VEL
LIN {X 0,Y 485.151,Z 243.055,A -85,B 0,C 180,E1 -6726.164,E2 -6726.164} C_VEL
LIN {X 0,Y 482.677,Z 243.358,A -85,B 0,C 180,E1 -6727.063,E2 -6727.063} C_VEL
LIN {X 0,Y 481.595,Z 243.583,A -85,B 0,C 180,E1 -6727.757,E2 -6727.757} C_VEL
LIN {X 0,Y 481.497,Z 243.73,A -85,B 0,C 180,E1 -6727.992,E2 -6727.992} C_VEL
LIN {X 0,Y 481.51,Z 244.902,A -85,B 0,C 180,E1 -6729.083,E2 -6729.083} C_VEL
LIN {X 0,Y 481.451,Z 249.431,A -85,B 0,C 180,E1 -6732.149,E2 -6732.149} C_VEL
LIN {X 0,Y 481.383,Z 253.357,A -85,B 0,C 180,E1 -6734.764,E2 -6734.764} C_VEL
LIN {X 0,Y 481.356,Z 258.602,A -85,B 0,C 180,E1 -6738.206,E2 -6738.206} C_VEL
LIN {X 0,Y 481.199,Z 263.89,A -85,B 0,C 180,E1 -6741.602,E2 -6741.602} C_VEL
LIN {X 0,Y 481.148,Z 267.885,A -85,B 0,C 180,E1 -6744.132,E2 -6744.132} C_VEL
LIN {X 0,Y 481.131,Z 271.885,A -85,B 0,C 180,E1 -6746.65,E2 -6746.65} C_VEL
LIN {X 0,Y 480.894,Z 274.314,A -85,B 0,C 180,E1 -6748.142,E2 -6748.142} C_VEL
LIN {X 0,Y 483.821,Z 288.962,A -85,B 0,C 180,E1 -6748.66,E2 -6748.66} C_VEL
LIN {X 0,Y 483.691,Z 299.782,A -85,B 0,C 180,E1 -6749.115,E2 -6749.115} C_VEL
LIN {X 0,Y 483.27,Z 312.017,A -85,B 0,C 180,E1 -6749.792,E2 -6749.792} C_VEL
LIN {X 0,Y 482.829,Z 323.523,A -85,B 0,C 180,E1 -6750.625,E2 -6750.625} C_VEL
LIN {X 0,Y 482.361,Z 333.903,A -85,B 0,C 180,E1 -6751.565,E2 -6751.565} C_VEL
LIN {X 0,Y 482.033,Z 342.392,A -85,B 0,C 180,E1 -6752.507,E2 -6752.507} C_VEL
LIN {X 0,Y 481.658,Z 350.254,A -85,B 0,C 180,E1 -6753.555,E2 -6753.555} C_VEL
LIN {X 0,Y 481.371,Z 357.954,A -85,B 0,C 180,E1 -6754.815,E2 -6754.815} C_VEL
LIN {X 0,Y 481.187,Z 364.327,A -85,B 0,C 180,E1 -6756.124,E2 -6756.124} C_VEL
LIN {X 0,Y 481.011,Z 369.773,A -85,B 0,C 180,E1 -6757.556,E2 -6757.556} C_VEL
LIN {X 0,Y 480.881,Z 373.413,A -85,B 0,C 180,E1 -6758.827,E2 -6758.827} C_VEL
LIN {X 0,Y 480.795,Z 376.036,A -85,B 0,C 180,E1 -6760.102,E2 -6760.102} C_VEL
LIN {X 0,Y 480.828,Z 377.985,A -85,B 0,C 180,E1 -6761.685,E2 -6761.685} C_VEL
LIN {X 0,Y 480.743,Z 378.443,A -85,B 0,C 180,E1 -6762.667,E2 -6762.667} C_VEL
LIN {X 0,Y 480.705,Z 378.427,A -85,B 0,C 180,E1 -6763.528,E2 -6763.528} C_VEL
LIN {X 0,Y 480.744,Z 378.007,A -85,B 0,C 180,E1 -6764.39,E2 -6764.39} C_VEL
LIN {X 0,Y 480.776,Z 377.124,A -85,B 0,C 180,E1 -6765.255,E2 -6765.255} C_VEL
LIN {X 0,Y 480.734,Z 375.818,A -85,B 0,C 180,E1 -6766.127,E2 -6766.127} C_VEL
LIN {X 0,Y 480.879,Z 373.012,A -85,B 0,C 180,E1 -6767.433,E2 -6767.433} C_VEL
LIN {X 0,Y 481.013,Z 369.091,A -85,B 0,C 180,E1 -6768.749,E2 -6768.749} C_VEL
LIN {X 0,Y 481.173,Z 363.927,A -85,B 0,C 180,E1 -6770.074,E2 -6770.074} C_VEL
LIN {X 0,Y 481.433,Z 357.326,A -85,B 0,C 180,E1 -6771.404,E2 -6771.404} C_VEL
LIN {X 0,Y 481.785,Z 348.919,A -85,B 0,C 180,E1 -6772.74,E2 -6772.74} C_VEL
LIN {X 0,Y 482.196,Z 339.376,A -85,B 0,C 180,E1 -6773.959,E2 -6773.959} C_VEL
LIN {X 0,Y 482.59,Z 329.371,A -85,B 0,C 180,E1 -6774.981,E2 -6774.981} C_VEL
LIN {X 0,Y 483.058,Z 318.454,A -85,B 0,C 180,E1 -6775.878,E2 -6775.878} C_VEL
LIN {X 0,Y 483.431,Z 308.198,A -85,B 0,C 180,E1 -6776.553,E2 -6776.553} C_VEL
LIN {X 0,Y 483.853,Z 297.233,A -85,B 0,C 180,E1 -6777.117,E2 -6777.117} C_VEL
LIN {X 0,Y 483.809,Z 288.477,A -85,B 0,C 180,E1 -6777.475,E2 -6777.475} C_VEL
LIN {X 0,Y 481.055,Z 275.383,A -85,B 0,C 180,E1 -6777.947,E2 -6777.947} C_VEL
LIN {X 0,Y 480.934,Z 274.387,A -85,B 0,C 180,E1 -6777.998,E2 -6777.998} C_VEL
LIN {X 0,Y 480.95,Z 270.02,A -85,B 0,C 180,E1 -6780.759,E2 -6780.759} C_VEL
LIN {X 0,Y 481.098,Z 265.418,A -85,B 0,C 180,E1 -6783.718,E2 -6783.718} C_VEL
LIN {X 0,Y 481.181,Z 260.753,A -85,B 0,C 180,E1 -6786.785,E2 -6786.785} C_VEL
LIN {X 0,Y 481.31,Z 256.998,A -85,B 0,C 180,E1 -6789.297,E2 -6789.297} C_VEL
LIN {X 0,Y 481.38,Z 252.79,A -85,B 0,C 180,E1 -6792.188,E2 -6792.188} C_VEL
LIN {X 0,Y 481.546,Z 249.512,A -85,B 0,C 180,E1 -6794.469,E2 -6794.469} C_VEL
LIN {X 0,Y 481.639,Z 246.199,A -85,B 0,C 180,E1 -6796.851,E2 -6796.851} C_VEL
LIN {X 0,Y 481.571,Z 243.504,A -85,B 0,C 180,E1 -6798.951,E2 -6798.951} C_VEL
LIN {X 0,Y 481.657,Z 243.494,A -85,B 0,C 180,E1 -6801.141,E2 -6801.141} C_VEL
LIN {X 0,Y 481.63,Z 243.496,A -85,B 0,C 180,E1 -6804.292,E2 -6804.292} C_VEL
LIN {X 0,Y 481.659,Z 243.493,A -85,B 0,C 180,E1 -6807.326,E2 -6807.326} C_VEL
LIN {X 0,Y 481.675,Z 243.489,A -85,B 0,C 180,E1 -6810.26,E2 -6810.26} C_VEL
LIN {X 0,Y 481.732,Z 243.48,A -85,B 0,C 180,E1 -6813.113,E2 -6813.113} C_VEL
LIN {X 0,Y 481.671,Z 243.486,A -85,B 0,C 180,E1 -6815.888,E2 -6815.888} C_VEL
LIN {X 0,Y 481.698,Z 243.484,A -85,B 0,C 180,E1 -6819.026,E2 -6819.026} C_VEL
LIN {X 0,Y 481.695,Z 243.484,A -85,B 0,C 180,E1 -6822.159,E2 -6822.159} C_VEL
LIN {X 0,Y 481.73,Z 243.478,A -85,B 0,C 180,E1 -6824.777,E2 -6824.777} C_VEL
LIN {X 0,Y 481.739,Z 243.479,A -85,B 0,C 180,E1 -6828.216,E2 -6828.216} C_VEL
LIN {X 0,Y 481.753,Z 243.478,A -85,B 0,C 180,E1 -6831.613,E2 -6831.613} C_VEL
LIN {X 0,Y 481.792,Z 243.471,A -85,B 0,C 180,E1 -6834.14,E2 -6834.14} C_VEL
LIN {X 0,Y 481.919,Z 243.458,A -85,B 0,C 180,E1 -6837.494,E2 -6837.494} C_VEL
LIN {X 0,Y 481.926,Z 243.453,A -85,B 0,C 180,E1 -6840.001,E2 -6840.001} C_VEL
LIN {X 0,Y 481.92,Z 243.455,A -85,B 0,C 180,E1 -6842.508,E2 -6842.508} C_VEL
LIN {X 0,Y 481.798,Z 243.469,A -85,B 0,C 180,E1 -6845.862,E2 -6845.862} C_VEL
LIN {X 0,Y 481.753,Z 243.477,A -85,B 0,C 180,E1 -6848.389,E2 -6848.389} C_VEL
LIN {X 0,Y 481.744,Z 243.476,A -85,B 0,C 180,E1 -6851.786,E2 -6851.786} C_VEL
LIN {X 0,Y 481.734,Z 243.48,A -85,B 0,C 180,E1 -6855.225,E2 -6855.225} C_VEL
LIN {X 0,Y 481.705,Z 243.486,A -85,B 0,C 180,E1 -6858.723,E2 -6858.723} C_VEL
LIN {X 0,Y 481.638,Z 243.493,A -85,B 0,C 180,E1 -6861.396,E2 -6861.396} C_VEL
LIN {X 0,Y 481.67,Z 243.488,A -85,B 0,C 180,E1 -6864.114,E2 -6864.114} C_VEL
LIN {X 0,Y 481.691,Z 243.486,A -85,B 0,C 180,E1 -6867.129,E2 -6867.129} C_VEL
LIN {X 0,Y 481.667,Z 243.488,A -85,B 0,C 180,E1 -6869.743,E2 -6869.743} C_VEL
LIN {X 0,Y 481.668,Z 243.487,A -85,B 0,C 180,E1 -6872.675,E2 -6872.675} C_VEL
LIN {X 0,Y 481.632,Z 243.491,A -85,B 0,C 180,E1 -6875.711,E2 -6875.711} C_VEL
LIN {X 0,Y 481.667,Z 243.486,A -85,B 0,C 180,E1 -6878.86,E2 -6878.86} C_VEL
LIN {X 0,Y 481.649,Z 243.488,A -85,B 0,C 180,E1 -6881.914,E2 -6881.914} C_VEL
LIN {X 0,Y 481.652,Z 243.485,A -85,B 0,C 180,E1 -6884.459,E2 -6884.459} C_VEL
LIN {X 0,Y 481.623,Z 243.496,A -85,B 0,C 180,E1 -6887.838,E2 -6887.838} C_VEL
LIN {X 0,Y 481.687,Z 243.562,A -85,B 0,C 180,E1 -6890.822,E2 -6890.822} C_VEL
LIN {X 0,Y 482.455,Z 248.269,A -85,B 0,C 180,E1 -6893.328,E2 -6893.328} C_VEL
LIN {X 0,Y 482.628,Z 252.416,A -85,B 0,C 180,E1 -6895.396,E2 -6895.396} C_VEL
LIN {X 0,Y 482.306,Z 258.747,A -85,B 0,C 180,E1 -6898.361,E2 -6898.361} C_VEL
LIN {X 0,Y 482.001,Z 265.16,A -85,B 0,C 180,E1 -6901.239,E2 -6901.239} C_VEL
LIN {X 0,Y 481.703,Z 273.333,A -85,B 0,C 180,E1 -6904.767,E2 -6904.767} C_VEL
LIN {X 0,Y 481.47,Z 280.357,A -85,B 0,C 180,E1 -6907.697,E2 -6907.697} C_VEL
LIN {X 0,Y 481.302,Z 286.944,A -85,B 0,C 180,E1 -6910.376,E2 -6910.376} C_VEL
LIN {X 0,Y 481.149,Z 294.66,A -85,B 0,C 180,E1 -6913.452,E2 -6913.452} C_VEL
LIN {X 0,Y 481.083,Z 298.659,A -85,B 0,C 180,E1 -6915.026,E2 -6915.026} C_VEL
LIN {X 0,Y 483.488,Z 314.25,A -85,B 0,C 180,E1 -6915.546,E2 -6915.546} C_VEL
LIN {X 0,Y 483.807,Z 318.239,A -85,B 0,C 180,E1 -6915.703,E2 -6915.703} C_VEL
LIN {X 0,Y 483.397,Z 329.817,A -85,B 0,C 180,E1 -6916.228,E2 -6916.228} C_VEL
LIN {X 0,Y 482.996,Z 340.976,A -85,B 0,C 180,E1 -6916.891,E2 -6916.891} C_VEL
LIN {X 0,Y 482.533,Z 351.422,A -85,B 0,C 180,E1 -6917.671,E2 -6917.671} C_VEL
LIN {X 0,Y 482.207,Z 361.969,A -85,B 0,C 180,E1 -6918.653,E2 -6918.653} C_VEL
LIN {X 0,Y 481.742,Z 371.135,A -85,B 0,C 180,E1 -6919.706,E2 -6919.706} C_VEL
LIN {X 0,Y 481.416,Z 380.075,A -85,B 0,C 180,E1 -6920.971,E2 -6920.971} C_VEL
LIN {X 0,Y 481.153,Z 387.277,A -85,B 0,C 180,E1 -6922.235,E2 -6922.235} C_VEL
LIN {X 0,Y 481.005,Z 393.012,A -85,B 0,C 180,E1 -6923.495,E2 -6923.495} C_VEL
LIN {X 0,Y 480.898,Z 398.182,A -85,B 0,C 180,E1 -6924.97,E2 -6924.97} C_VEL
LIN {X 0,Y 480.828,Z 400.481,A -85,B 0,C 180,E1 -6925.809,E2 -6925.809} C_VEL
LIN {X 0,Y 480.889,Z 402.347,A -85,B 0,C 180,E1 -6926.649,E2 -6926.649} C_VEL
LIN {X 0,Y 480.793,Z 404.743,A -85,B 0,C 180,E1 -6928.325,E2 -6928.325} C_VEL
LIN {X 0,Y 480.76,Z 405.353,A -85,B 0,C 180,E1 -6929.162,E2 -6929.162} C_VEL
LIN {X 0,Y 480.743,Z 405.571,A -85,B 0,C 180,E1 -6930,E2 -6930} C_VEL
LIN {X 0,Y 480.793,Z 404.752,A -85,B 0,C 180,E1 -6931.675,E2 -6931.675} C_VEL
LIN {X 0,Y 480.824,Z 403.759,A -85,B 0,C 180,E1 -6932.513,E2 -6932.513} C_VEL
LIN {X 0,Y 480.889,Z 402.365,A -85,B 0,C 180,E1 -6933.351,E2 -6933.351} C_VEL
LIN {X 0,Y 480.84,Z 399.428,A -85,B 0,C 180,E1 -6934.611,E2 -6934.611} C_VEL
LIN {X 0,Y 480.931,Z 395.454,A -85,B 0,C 180,E1 -6935.871,E2 -6935.871} C_VEL
LIN {X 0,Y 481.113,Z 389.34,A -85,B 0,C 180,E1 -6937.343,E2 -6937.343} C_VEL
LIN {X 0,Y 481.325,Z 382.658,A -85,B 0,C 180,E1 -6938.607,E2 -6938.607} C_VEL
LIN {X 0,Y 481.62,Z 374.366,A -85,B 0,C 180,E1 -6939.873,E2 -6939.873} C_VEL
LIN {X 0,Y 482.018,Z 365.865,A -85,B 0,C 180,E1 -6940.926,E2 -6940.926} C_VEL
LIN {X 0,Y 482.438,Z 355.375,A -85,B 0,C 180,E1 -6941.979,E2 -6941.979} C_VEL
LIN {X 0,Y 482.847,Z 343.946,A -85,B 0,C 180,E1 -6942.899,E2 -6942.899} C_VEL
LIN {X 0,Y 483.336,Z 331.594,A -85,B 0,C 180,E1 -6943.667,E2 -6943.667} C_VEL
LIN {X 0,Y 483.759,Z 319.193,A -85,B 0,C 180,E1 -6944.245,E2 -6944.245} C_VEL
LIN {X 0,Y 483.501,Z 314.548,A -85,B 0,C 180,E1 -6944.427,E2 -6944.427} C_VEL
LIN {X 0,Y 481.478,Z 301.589,A -85,B 0,C 180,E1 -6944.857,E2 -6944.857} C_VEL
LIN {X 0,Y 481.064,Z 298.751,A -85,B 0,C 180,E1 -6944.948,E2 -6944.948} C_VEL
LIN {X 0,Y 481.189,Z 291.322,A -85,B 0,C 180,E1 -6947.861,E2 -6947.861} C_VEL
LIN {X 0,Y 481.417,Z 283.718,A -85,B 0,C 180,E1 -6950.882,E2 -6950.882} C_VEL
LIN {X 0,Y 481.566,Z 275.725,A -85,B 0,C 180,E1 -6954.118,E2 -6954.118} C_VEL
LIN {X 0,Y 481.796,Z 268.406,A -85,B 0,C 180,E1 -6957.149,E2 -6957.149} C_VEL
LIN {X 0,Y 482.03,Z 261.254,A -85,B 0,C 180,E1 -6960.192,E2 -6960.192} C_VEL
LIN {X 0,Y 482.299,Z 254.554,A -85,B 0,C 180,E1 -6963.123,E2 -6963.123} C_VEL
LIN {X 0,Y 482.447,Z 248.99,A -85,B 0,C 180,E1 -6965.639,E2 -6965.639} C_VEL
LIN {X 0,Y 481.733,Z 243.723,A -85,B 0,C 180,E1 -6968.174,E2 -6968.174} C_VEL
LIN {X 0,Y 481.675,Z 243.489,A -85,B 0,C 180,E1 -6968.858,E2 -6968.858} C_VEL
LIN {X 0,Y 481.612,Z 243.492,A -85,B 0,C 180,E1 -6972.163,E2 -6972.163} C_VEL
LIN {X 0,Y 481.647,Z 243.488,A -85,B 0,C 180,E1 -6974.458,E2 -6974.458} C_VEL
LIN {X 0,Y 481.61,Z 243.491,A -85,B 0,C 180,E1 -6977.834,E2 -6977.834} C_VEL
LIN {X 0,Y 481.642,Z 243.493,A -85,B 0,C 180,E1 -6980.655,E2 -6980.655} C_VEL
LIN {X 0,Y 481.602,Z 243.492,A -85,B 0,C 180,E1 -6983.379,E2 -6983.379} C_VEL
LIN {X 0,Y 481.672,Z 243.489,A -85,B 0,C 180,E1 -6986.326,E2 -6986.326} C_VEL
LIN {X 0,Y 481.643,Z 243.488,A -85,B 0,C 180,E1 -6989.417,E2 -6989.417} C_VEL
LIN {X 0,Y 481.651,Z 243.492,A -85,B 0,C 180,E1 -6992.164,E2 -6992.164} C_VEL
LIN {X 0,Y 481.672,Z 243.484,A -85,B 0,C 180,E1 -6994.967,E2 -6994.967} C_VEL
LIN {X 0,Y 481.641,Z 243.491,A -85,B 0,C 180,E1 -6997.703,E2 -6997.703} C_VEL
LIN {X 0,Y 481.697,Z 243.481,A -85,B 0,C 180,E1 -7000.392,E2 -7000.392} C_VEL
LIN {X 0,Y 481.672,Z 243.486,A -85,B 0,C 180,E1 -7003.032,E2 -7003.032} C_VEL
LIN {X 0,Y 481.681,Z 243.487,A -85,B 0,C 180,E1 -7005.638,E2 -7005.638} C_VEL
LIN {X 0,Y 481.742,Z 243.476,A -85,B 0,C 180,E1 -7008.214,E2 -7008.214} C_VEL
LIN {X 0,Y 481.754,Z 243.477,A -85,B 0,C 180,E1 -7011.611,E2 -7011.611} C_VEL
LIN {X 0,Y 481.806,Z 243.468,A -85,B 0,C 180,E1 -7014.139,E2 -7014.139} C_VEL
LIN {X 0,Y 481.918,Z 243.455,A -85,B 0,C 180,E1 -7017.492,E2 -7017.492} C_VEL
LIN {X 0,Y 481.929,Z 243.453,A -85,B 0,C 180,E1 -7019.999,E2 -7019.999} C_VEL
LIN {X 0,Y 481.918,Z 243.457,A -85,B 0,C 180,E1 -7022.506,E2 -7022.506} C_VEL
LIN {X 0,Y 481.812,Z 243.468,A -85,B 0,C 180,E1 -7025.859,E2 -7025.859} C_VEL
LIN {X 0,Y 481.754,Z 243.477,A -85,B 0,C 180,E1 -7028.387,E2 -7028.387} C_VEL
LIN {X 0,Y 481.742,Z 243.477,A -85,B 0,C 180,E1 -7031.784,E2 -7031.784} C_VEL
LIN {X 0,Y 481.731,Z 243.477,A -85,B 0,C 180,E1 -7035.223,E2 -7035.223} C_VEL
LIN {X 0,Y 481.701,Z 243.481,A -85,B 0,C 180,E1 -7038.721,E2 -7038.721} C_VEL
LIN {X 0,Y 481.635,Z 243.49,A -85,B 0,C 180,E1 -7041.394,E2 -7041.394} C_VEL
LIN {X 0,Y 481.665,Z 243.486,A -85,B 0,C 180,E1 -7044.112,E2 -7044.112} C_VEL
LIN {X 0,Y 481.74,Z 243.477,A -85,B 0,C 180,E1 -7047.14,E2 -7047.14} C_VEL
LIN {X 0,Y 481.676,Z 243.486,A -85,B 0,C 180,E1 -7049.74,E2 -7049.74} C_VEL
LIN {X 0,Y 481.661,Z 243.485,A -85,B 0,C 180,E1 -7052.674,E2 -7052.674} C_VEL
LIN {X 0,Y 481.631,Z 243.489,A -85,B 0,C 180,E1 -7055.708,E2 -7055.708} C_VEL
LIN {X 0,Y 481.707,Z 243.481,A -85,B 0,C 180,E1 -7059.354,E2 -7059.354} C_VEL
LIN {X 0,Y 481.662,Z 243.483,A -85,B 0,C 180,E1 -7062.157,E2 -7062.157} C_VEL
LIN {X 0,Y 481.647,Z 243.488,A -85,B 0,C 180,E1 -7064.457,E2 -7064.457} C_VEL
LIN {X 0,Y 481.641,Z 243.485,A -85,B 0,C 180,E1 -7067.84,E2 -7067.84} C_VEL
LIN {X 0,Y 481.668,Z 243.49,A -85,B 0,C 180,E1 -7070.651,E2 -7070.651} C_VEL
LIN {X 0,Y 481.617,Z 243.489,A -85,B 0,C 180,E1 -7073.376,E2 -7073.376} C_VEL
LIN {X 0,Y 481.697,Z 243.485,A -85,B 0,C 180,E1 -7076.33,E2 -7076.33} C_VEL
LIN {X 0,Y 481.637,Z 243.487,A -85,B 0,C 180,E1 -7079.417,E2 -7079.417} C_VEL
LIN {X 0,Y 481.68,Z 243.488,A -85,B 0,C 180,E1 -7082.168,E2 -7082.168} C_VEL
LIN {X 0,Y 481.676,Z 243.483,A -85,B 0,C 180,E1 -7084.968,E2 -7084.968} C_VEL
LIN {X 0,Y 481.523,Z 243.505,A -85,B 0,C 180,E1 -7087.699,E2 -7087.699} C_VEL
LIN {X 0,Y 481.497,Z 243.73,A -85,B 0,C 180,E1 -7087.992,E2 -7087.992} C_VEL
LIN {X 0,Y 480.809,Z 244.498,A -85,B 0,C 180,E1 -7088.684,E2 -7088.684} C_VEL
LIN {X 0,Y 477.965,Z 246.361,A -85,B 0,C 180,E1 -7089.798,E2 -7089.798} C_VEL
LIN {X 0,Y 475.566,Z 247.945,A -85,B 0,C 180,E1 -7090.692,E2 -7090.692} C_VEL
LIN {X 0,Y 474.528,Z 249.074,A -85,B 0,C 180,E1 -7091.384,E2 -7091.384} C_VEL
LIN {X 0,Y 474.438,Z 249.428,A -85,B 0,C 180,E1 -7091.619,E2 -7091.619} C_VEL
LIN {X 0,Y 474.337,Z 253.743,A -85,B 0,C 180,E1 -7094.533,E2 -7094.533} C_VEL
LIN {X 0,Y 474.288,Z 259.006,A -85,B 0,C 180,E1 -7098.027,E2 -7098.027} C_VEL
LIN {X 0,Y 474.143,Z 264.323,A -85,B 0,C 180,E1 -7101.476,E2 -7101.476} C_VEL
LIN {X 0,Y 474.094,Z 268.319,A -85,B 0,C 180,E1 -7104.044,E2 -7104.044} C_VEL
LIN {X 0,Y 474.079,Z 272.367,A -85,B 0,C 180,E1 -7106.601,E2 -7106.601} C_VEL
LIN {X 0,Y 473.838,Z 274.498,A -85,B 0,C 180,E1 -7107.928,E2 -7107.928} C_VEL
LIN {X 0,Y 476.869,Z 289.474,A -85,B 0,C 180,E1 -7108.469,E2 -7108.469} C_VEL
LIN {X 0,Y 476.922,Z 297.098,A -85,B 0,C 180,E1 -7108.786,E2 -7108.786} C_VEL
LIN {X 0,Y 476.509,Z 308.273,A -85,B 0,C 180,E1 -7109.366,E2 -7109.366} C_VEL
LIN {X 0,Y 475.997,Z 320.737,A -85,B 0,C 180,E1 -7110.211,E2 -7110.211} C_VEL
LIN {X 0,Y 475.518,Z 331.698,A -85,B 0,C 180,E1 -7111.164,E2 -7111.164} C_VEL
LIN {X 0,Y 475.049,Z 342.361,A -85,B 0,C 180,E1 -7112.332,E2 -7112.332} C_VEL
LIN {X 0,Y 474.626,Z 350.27,A -85,B 0,C 180,E1 -7113.395,E2 -7113.395} C_VEL
LIN {X 0,Y 474.321,Z 358.018,A -85,B 0,C 180,E1 -7114.674,E2 -7114.674} C_VEL
LIN {X 0,Y 474.142,Z 364.22,A -85,B 0,C 180,E1 -7115.955,E2 -7115.955} C_VEL
LIN {X 0,Y 473.976,Z 369.172,A -85,B 0,C 180,E1 -7117.24,E2 -7117.24} C_VEL
LIN {X 0,Y 473.83,Z 373.012,A -85,B 0,C 180,E1 -7118.53,E2 -7118.53} C_VEL
LIN {X 0,Y 473.73,Z 374.996,A -85,B 0,C 180,E1 -7119.392,E2 -7119.392} C_VEL
LIN {X 0,Y 473.707,Z 376.56,A -85,B 0,C 180,E1 -7120.255,E2 -7120.255} C_VEL
LIN {X 0,Y 473.718,Z 378.223,A -85,B 0,C 180,E1 -7121.724,E2 -7121.724} C_VEL
LIN {X 0,Y 473.647,Z 378.68,A -85,B 0,C 180,E1 -7122.86,E2 -7122.86} C_VEL
LIN {X 0,Y 473.61,Z 378.586,A -85,B 0,C 180,E1 -7123.734,E2 -7123.734} C_VEL
LIN {X 0,Y 473.695,Z 377.257,A -85,B 0,C 180,E1 -7125.345,E2 -7125.345} C_VEL
LIN {X 0,Y 473.666,Z 375.688,A -85,B 0,C 180,E1 -7126.374,E2 -7126.374} C_VEL
LIN {X 0,Y 473.841,Z 372.727,A -85,B 0,C 180,E1 -7127.701,E2 -7127.701} C_VEL
LIN {X 0,Y 473.974,Z 368.638,A -85,B 0,C 180,E1 -7129.038,E2 -7129.038} C_VEL
LIN {X 0,Y 474.161,Z 362.208,A -85,B 0,C 180,E1 -7130.61,E2 -7130.61} C_VEL
LIN {X 0,Y 474.487,Z 355.103,A -85,B 0,C 180,E1 -7131.962,E2 -7131.962} C_VEL
LIN {X 0,Y 474.909,Z 346.851,A -85,B 0,C 180,E1 -7133.215,E2 -7133.215} C_VEL
LIN {X 0,Y 475.294,Z 337.694,A -85,B 0,C 180,E1 -7134.341,E2 -7134.341} C_VEL
LIN {X 0,Y 475.797,Z 327.441,A -85,B 0,C 180,E1 -7135.363,E2 -7135.363} C_VEL
LIN {X 0,Y 476.228,Z 317.101,A -85,B 0,C 180,E1 -7136.196,E2 -7136.196} C_VEL
LIN {X 0,Y 476.695,Z 304.985,A -85,B 0,C 180,E1 -7136.958,E2 -7136.958} C_VEL
LIN {X 0,Y 477.116,Z 292.859,A -85,B 0,C 180,E1 -7137.532,E2 -7137.532} C_VEL
LIN {X 0,Y 476.771,Z 288.607,A -85,B 0,C 180,E1 -7137.709,E2 -7137.709} C_VEL
LIN {X 0,Y 474.089,Z 275.945,A -85,B 0,C 180,E1 -7138.179,E2 -7138.179} C_VEL
LIN {X 0,Y 473.863,Z 274.613,A -85,B 0,C 180,E1 -7138.227,E2 -7138.227} C_VEL
LIN {X 0,Y 473.914,Z 269.871,A -85,B 0,C 180,E1 -7141.267,E2 -7141.267} C_VEL
LIN {X 0,Y 474.048,Z 265.251,A -85,B 0,C 180,E1 -7144.288,E2 -7144.288} C_VEL
LIN {X 0,Y 474.178,Z 260.562,A -85,B 0,C 180,E1 -7147.421,E2 -7147.421} C_VEL
LIN {X 0,Y 474.263,Z 257.367,A -85,B 0,C 180,E1 -7149.597,E2 -7149.597} C_VEL
LIN {X 0,Y 474.39,Z 252.559,A -85,B 0,C 180,E1 -7152.958,E2 -7152.958} C_VEL
LIN {X 0,Y 474.566,Z 248.463,A -85,B 0,C 180,E1 -7155.892,E2 -7155.892} C_VEL
LIN {X 0,Y 474.576,Z 245.321,A -85,B 0,C 180,E1 -7158.212,E2 -7158.212} C_VEL
LIN {X 0,Y 474.561,Z 244.378,A -85,B 0,C 180,E1 -7159.049,E2 -7159.049} C_VEL
LIN {X 0,Y 474.597,Z 244.369,A -85,B 0,C 180,E1 -7161.704,E2 -7161.704} C_VEL
LIN {X 0,Y 474.617,Z 244.367,A -85,B 0,C 180,E1 -7164.727,E2 -7164.727} C_VEL
LIN {X 0,Y 474.623,Z 244.366,A -85,B 0,C 180,E1 -7167.788,E2 -7167.788} C_VEL
LIN {X 0,Y 474.619,Z 244.364,A -85,B 0,C 180,E1 -7170.883,E2 -7170.883} C_VEL
LIN {X 0,Y 474.647,Z 244.362,A -85,B 0,C 180,E1 -7173.629,E2 -7173.629} C_VEL
LIN {X 0,Y 474.629,Z 244.363,A -85,B 0,C 180,E1 -7176.64,E2 -7176.64} C_VEL
LIN {X 0,Y 474.664,Z 244.361,A -85,B 0,C 180,E1 -7179.186,E2 -7179.186} C_VEL
LIN {X 0,Y 474.645,Z 244.361,A -85,B 0,C 180,E1 -7181.885,E2 -7181.885} C_VEL
LIN {X 0,Y 474.687,Z 244.355,A -85,B 0,C 180,E1 -7184.545,E2 -7184.545} C_VEL
LIN {X 0,Y 474.692,Z 244.356,A -85,B 0,C 180,E1 -7188.038,E2 -7188.038} C_VEL
LIN {X 0,Y 474.718,Z 244.355,A -85,B 0,C 180,E1 -7191.487,E2 -7191.487} C_VEL
LIN {X 0,Y 474.755,Z 244.347,A -85,B 0,C 180,E1 -7194.053,E2 -7194.053} C_VEL
LIN {X 0,Y 474.886,Z 244.334,A -85,B 0,C 180,E1 -7197.456,E2 -7197.456} C_VEL
LIN {X 0,Y 474.897,Z 244.329,A -85,B 0,C 180,E1 -7200.001,E2 -7200.001} C_VEL
LIN {X 0,Y 474.886,Z 244.331,A -85,B 0,C 180,E1 -7202.546,E2 -7202.546} C_VEL
LIN {X 0,Y 474.76,Z 244.345,A -85,B 0,C 180,E1 -7205.949,E2 -7205.949} C_VEL
LIN {X 0,Y 474.719,Z 244.352,A -85,B 0,C 180,E1 -7208.515,E2 -7208.515} C_VEL
LIN {X 0,Y 474.697,Z 244.354,A -85,B 0,C 180,E1 -7211.964,E2 -7211.964} C_VEL
LIN {X 0,Y 474.692,Z 244.359,A -85,B 0,C 180,E1 -7215.457,E2 -7215.457} C_VEL
LIN {X 0,Y 474.657,Z 244.362,A -85,B 0,C 180,E1 -7219.011,E2 -7219.011} C_VEL
LIN {X 0,Y 474.582,Z 244.374,A -85,B 0,C 180,E1 -7221.73,E2 -7221.73} C_VEL
LIN {X 0,Y 474.652,Z 244.365,A -85,B 0,C 180,E1 -7224.494,E2 -7224.494} C_VEL
LIN {X 0,Y 474.631,Z 244.367,A -85,B 0,C 180,E1 -7227.325,E2 -7227.325} C_VEL
LIN {X 0,Y 474.598,Z 244.369,A -85,B 0,C 180,E1 -7230.232,E2 -7230.232} C_VEL
LIN {X 0,Y 474.638,Z 244.363,A -85,B 0,C 180,E1 -7233.221,E2 -7233.221} C_VEL
LIN {X 0,Y 474.584,Z 244.37,A -85,B 0,C 180,E1 -7236.325,E2 -7236.325} C_VEL
LIN {X 0,Y 474.625,Z 244.366,A -85,B 0,C 180,E1 -7239.649,E2 -7239.649} C_VEL
LIN {X 0,Y 474.612,Z 244.368,A -85,B 0,C 180,E1 -7242.935,E2 -7242.935} C_VEL
LIN {X 0,Y 474.599,Z 244.371,A -85,B 0,C 180,E1 -7245.895,E2 -7245.895} C_VEL
LIN {X 0,Y 474.6,Z 244.371,A -85,B 0,C 180,E1 -7249.046,E2 -7249.046} C_VEL
LIN {X 0,Y 474.655,Z 244.518,A -85,B 0,C 180,E1 -7250.594,E2 -7250.594} C_VEL
LIN {X 0,Y 475.375,Z 248.883,A -85,B 0,C 180,E1 -7252.973,E2 -7252.973} C_VEL
LIN {X 0,Y 475.65,Z 253.522,A -85,B 0,C 180,E1 -7255.33,E2 -7255.33} C_VEL
LIN {X 0,Y 475.307,Z 259.811,A -85,B 0,C 180,E1 -7258.339,E2 -7258.339} C_VEL
LIN {X 0,Y 474.977,Z 266.229,A -85,B 0,C 180,E1 -7261.263,E2 -7261.263} C_VEL
LIN {X 0,Y 474.656,Z 273.779,A -85,B 0,C 180,E1 -7264.583,E2 -7264.583} C_VEL
LIN {X 0,Y 474.408,Z 281.363,A -85,B 0,C 180,E1 -7267.805,E2 -7267.805} C_VEL
LIN {X 0,Y 474.219,Z 287.923,A -85,B 0,C 180,E1 -7270.522,E2 -7270.522} C_VEL
LIN {X 0,Y 474.071,Z 295.614,A -85,B 0,C 180,E1 -7273.64,E2 -7273.64} C_VEL
LIN {X 0,Y 474.016,Z 298.51,A -85,B 0,C 180,E1 -7274.797,E2 -7274.797} C_VEL
LIN {X 0,Y 476.246,Z 312.502,A -85,B 0,C 180,E1 -7275.253,E2 -7275.253} C_VEL
LIN {X 0,Y 476.903,Z 319.61,A -85,B 0,C 180,E1 -7275.546,E2 -7275.546} C_VEL
LIN {X 0,Y 476.421,Z 331.799,A -85,B 0,C 180,E1 -7276.131,E2 -7276.131} C_VEL
LIN {X 0,Y 475.945,Z 343.552,A -85,B 0,C 180,E1 -7276.878,E2 -7276.878} C_VEL
LIN {X 0,Y 475.502,Z 354.632,A -85,B 0,C 180,E1 -7277.78,E2 -7277.78} C_VEL
LIN {X 0,Y 475.139,Z 363.798,A -85,B 0,C 180,E1 -7278.698,E2 -7278.698} C_VEL
LIN {X 0,Y 474.63,Z 372.621,A -85,B 0,C 180,E1 -7279.765,E2 -7279.765} C_VEL
LIN {X 0,Y 474.315,Z 381.232,A -85,B 0,C 180,E1 -7281.05,E2 -7281.05} C_VEL
LIN {X 0,Y 474.046,Z 388.126,A -85,B 0,C 180,E1 -7282.332,E2 -7282.332} C_VEL
LIN {X 0,Y 473.906,Z 393.301,A -85,B 0,C 180,E1 -7283.521,E2 -7283.521} C_VEL
LIN {X 0,Y 473.829,Z 397.992,A -85,B 0,C 180,E1 -7284.894,E2 -7284.894} C_VEL
LIN {X 0,Y 473.735,Z 400.288,A -85,B 0,C 180,E1 -7285.746,E2 -7285.746} C_VEL
LIN {X 0,Y 473.796,Z 402.152,A -85,B 0,C 180,E1 -7286.599,E2 -7286.599} C_VEL
LIN {X 0,Y 473.742,Z 403.548,A -85,B 0,C 180,E1 -7287.449,E2 -7287.449} C_VEL
LIN {X 0,Y 473.689,Z 405.155,A -85,B 0,C 180,E1 -7289.15,E2 -7289.15} C_VEL
LIN {X 0,Y 473.67,Z 405.372,A -85,B 0,C 180,E1 -7290,E2 -7290} C_VEL
LIN {X 0,Y 473.689,Z 405.156,A -85,B 0,C 180,E1 -7290.85,E2 -7290.85} C_VEL
LIN {X 0,Y 473.742,Z 403.556,A -85,B 0,C 180,E1 -7292.551,E2 -7292.551} C_VEL
LIN {X 0,Y 473.796,Z 402.16,A -85,B 0,C 180,E1 -7293.402,E2 -7293.402} C_VEL
LIN {X 0,Y 473.763,Z 399.22,A -85,B 0,C 180,E1 -7294.68,E2 -7294.68} C_VEL
LIN {X 0,Y 473.839,Z 395.24,A -85,B 0,C 180,E1 -7295.959,E2 -7295.959} C_VEL
LIN {X 0,Y 474.025,Z 389.116,A -85,B 0,C 180,E1 -7297.454,E2 -7297.454} C_VEL
LIN {X 0,Y 474.288,Z 382.425,A -85,B 0,C 180,E1 -7298.736,E2 -7298.736} C_VEL
LIN {X 0,Y 474.588,Z 374.12,A -85,B 0,C 180,E1 -7300.02,E2 -7300.02} C_VEL
LIN {X 0,Y 475.004,Z 365.599,A -85,B 0,C 180,E1 -7301.089,E2 -7301.089} C_VEL
LIN {X 0,Y 475.44,Z 355.284,A -85,B 0,C 180,E1 -7302.139,E2 -7302.139} C_VEL
LIN {X 0,Y 475.918,Z 343.628,A -85,B 0,C 180,E1 -7303.09,E2 -7303.09} C_VEL
LIN {X 0,Y 476.427,Z 331.218,A -85,B 0,C 180,E1 -7303.869,E2 -7303.869} C_VEL
LIN {X 0,Y 476.844,Z 318.751,A -85,B 0,C 180,E1 -7304.456,E2 -7304.456} C_VEL
LIN {X 0,Y 475.433,Z 307.472,A -85,B 0,C 180,E1 -7304.885,E2 -7304.885} C_VEL
LIN {X 0,Y 474.015,Z 298.61,A -85,B 0,C 180,E1 -7305.148,E2 -7305.148} C_VEL
LIN {X 0,Y 474.163,Z 290.335,A -85,B 0,C 180,E1 -7308.448,E2 -7308.448} C_VEL
LIN {X 0,Y 474.4,Z 282.218,A -85,B 0,C 180,E1 -7311.737,E2 -7311.737} C_VEL
LIN {X 0,Y 474.589,Z 274.444,A -85,B 0,C 180,E1 -7314.951,E2 -7314.951} C_VEL
LIN {X 0,Y 474.775,Z 267.728,A -85,B 0,C 180,E1 -7317.792,E2 -7317.792} C_VEL
LIN {X 0,Y 475.052,Z 260.575,A -85,B 0,C 180,E1 -7320.899,E2 -7320.899} C_VEL
LIN {X 0,Y 475.378,Z 253.255,A -85,B 0,C 180,E1 -7324.179,E2 -7324.179} C_VEL
LIN {X 0,Y 475.317,Z 248.797,A -85,B 0,C 180,E1 -7326.258,E2 -7326.258} C_VEL
LIN {X 0,Y 474.652,Z 244.364,A -85,B 0,C 180,E1 -7328.452,E2 -7328.452} C_VEL
LIN {X 0,Y 474.589,Z 244.366,A -85,B 0,C 180,E1 -7331.788,E2 -7331.788} C_VEL
LIN {X 0,Y 474.596,Z 244.366,A -85,B 0,C 180,E1 -7335.299,E2 -7335.299} C_VEL
LIN {X 0,Y 474.587,Z 244.367,A -85,B 0,C 180,E1 -7338.21,E2 -7338.21} C_VEL
LIN {X 0,Y 474.612,Z 244.367,A -85,B 0,C 180,E1 -7340.45,E2 -7340.45} C_VEL
LIN {X 0,Y 474.565,Z 244.369,A -85,B 0,C 180,E1 -7343.674,E2 -7343.674} C_VEL
LIN {X 0,Y 474.621,Z 244.364,A -85,B 0,C 180,E1 -7346.777,E2 -7346.777} C_VEL
LIN {X 0,Y 474.594,Z 244.367,A -85,B 0,C 180,E1 -7349.768,E2 -7349.768} C_VEL
LIN {X 0,Y 474.631,Z 244.362,A -85,B 0,C 180,E1 -7352.675,E2 -7352.675} C_VEL
LIN {X 0,Y 474.624,Z 244.364,A -85,B 0,C 180,E1 -7355.504,E2 -7355.504} C_VEL
LIN {X 0,Y 474.628,Z 244.362,A -85,B 0,C 180,E1 -7358.883,E2 -7358.883} C_VEL
LIN {X 0,Y 474.639,Z 244.364,A -85,B 0,C 180,E1 -7361.883,E2 -7361.883} C_VEL
LIN {X 0,Y 474.692,Z 244.354,A -85,B 0,C 180,E1 -7364.543,E2 -7364.543} C_VEL
LIN {X 0,Y 474.696,Z 244.354,A -85,B 0,C 180,E1 -7368.036,E2 -7368.036} C_VEL
LIN {X 0,Y 474.719,Z 244.354,A -85,B 0,C 180,E1 -7371.485,E2 -7371.485} C_VEL
LIN {X 0,Y 474.769,Z 244.344,A -85,B 0,C 180,E1 -7374.051,E2 -7374.051} C_VEL
LIN {X 0,Y 474.884,Z 244.332,A -85,B 0,C 180,E1 -7377.454,E2 -7377.454} C_VEL
LIN {X 0,Y 474.868,Z 244.334,A -85,B 0,C 180,E1 -7380.847,E2 -7380.847} C_VEL
LIN {X 0,Y 474.885,Z 244.333,A -85,B 0,C 180,E1 -7382.544,E2 -7382.544} C_VEL
LIN {X 0,Y 474.774,Z 244.345,A -85,B 0,C 180,E1 -7385.947,E2 -7385.947} C_VEL
LIN {X 0,Y 474.719,Z 244.353,A -85,B 0,C 180,E1 -7388.513,E2 -7388.513} C_VEL
LIN {X 0,Y 474.695,Z 244.357,A -85,B 0,C 180,E1 -7391.962,E2 -7391.962} C_VEL
LIN {X 0,Y 474.688,Z 244.355,A -85,B 0,C 180,E1 -7395.455,E2 -7395.455} C_VEL
LIN {X 0,Y 474.654,Z 244.358,A -85,B 0,C 180,E1 -7399.009,E2 -7399.009} C_VEL
LIN {X 0,Y 474.579,Z 244.372,A -85,B 0,C 180,E1 -7401.728,E2 -7401.728} C_VEL
LIN {X 0,Y 474.647,Z 244.359,A -85,B 0,C 180,E1 -7404.492,E2 -7404.492} C_VEL
LIN {X 0,Y 474.687,Z 244.358,A -85,B 0,C 180,E1 -7407.338,E2 -7407.338} C_VEL
LIN {X 0,Y 474.597,Z 244.365,A -85,B 0,C 180,E1 -7410.811,E2 -7410.811} C_VEL
LIN {X 0,Y 474.626,Z 244.361,A -85,B 0,C 180,E1 -7413.983,E2 -7413.983} C_VEL
LIN {X 0,Y 474.565,Z 244.372,A -85,B 0,C 180,E1 -7416.9,E2 -7416.9} C_VEL
LIN {X 0,Y 474.642,Z 244.359,A -85,B 0,C 180,E1 -7419.651,E2 -7419.651} C_VEL
LIN {X 0,Y 474.639,Z 244.366,A -85,B 0,C 180,E1 -7422.93,E2 -7422.93} C_VEL
LIN {X 0,Y 474.602,Z 244.362,A -85,B 0,C 180,E1 -7425.895,E2 -7425.895} C_VEL
LIN {X 0,Y 474.619,Z 244.364,A -85,B 0,C 180,E1 -7429.04,E2 -7429.04} C_VEL
LIN {X 0,Y 474.597,Z 244.363,A -85,B 0,C 180,E1 -7431.704,E2 -7431.704} C_VEL
LIN {X 0,Y 474.616,Z 244.366,A -85,B 0,C 180,E1 -7434.726,E2 -7434.726} C_VEL
LIN {X 0,Y 474.623,Z 244.362,A -85,B 0,C 180,E1 -7437.788,E2 -7437.788} C_VEL
LIN {X 0,Y 474.61,Z 244.363,A -85,B 0,C 180,E1 -7440.885,E2 -7440.885} C_VEL
LIN {X 0,Y 474.617,Z 244.364,A -85,B 0,C 180,E1 -7443.626,E2 -7443.626} C_VEL
LIN {X 0,Y 474.568,Z 244.369,A -85,B 0,C 180,E1 -7446.657,E2 -7446.657} C_VEL
LIN {X 0,Y 474.431,Z 244.558,A -85,B 0,C 180,E1 -7448.264,E2 -7448.264} C_VEL
LIN {X 0,Y 474.438,Z 249.428,A -85,B 0,C 180,E1 -7451.619,E2 -7451.619} C_VEL
LIN {X 0,Y 473.751,Z 250.529,A -85,B 0,C 180,E1 -7452.314,E2 -7452.314} C_VEL
LIN {X 0,Y 470.856,Z 252.509,A -85,B 0,C 180,E1 -7453.438,E2 -7453.438} C_VEL
LIN {X 0,Y 468.399,Z 254.108,A -85,B 0,C 180,E1 -7454.344,E2 -7454.344} C_VEL
LIN {X 0,Y 467.321,Z 255.252,A -85,B 0,C 180,E1 -7455.046,E2 -7455.046} C_VEL
LIN {X 0,Y 467.221,Z 255.612,A -85,B 0,C 180,E1 -7455.284,E2 -7455.284} C_VEL
LIN {X 0,Y 467.226,Z 259.481,A -85,B 0,C 180,E1 -7457.877,E2 -7457.877} C_VEL
LIN {X 0,Y 467.063,Z 264.757,A -85,B 0,C 180,E1 -7461.346,E2 -7461.346} C_VEL
LIN {X 0,Y 467.043,Z 268.773,A -85,B 0,C 180,E1 -7463.954,E2 -7463.954} C_VEL
LIN {X 0,Y 466.998,Z 272.834,A -85,B 0,C 180,E1 -7466.549,E2 -7466.549} C_VEL
LIN {X 0,Y 466.795,Z 274.67,A -85,B 0,C 180,E1 -7467.708,E2 -7467.708} C_VEL
LIN {X 0,Y 469.933,Z 290.237,A -85,B 0,C 180,E1 -7468.286,E2 -7468.286} C_VEL
LIN {X 0,Y 470.019,Z 297.699,A -85,B 0,C 180,E1 -7468.608,E2 -7468.608} C_VEL
LIN {X 0,Y 469.549,Z 309.667,A -85,B 0,C 180,E1 -7469.25,E2 -7469.25} C_VEL
LIN {X 0,Y 469.071,Z 320.501,A -85,B 0,C 180,E1 -7470,E2 -7470} C_VEL
LIN {X 0,Y 468.578,Z 331.572,A -85,B 0,C 180,E1 -7470.967,E2 -7470.967} C_VEL
LIN {X 0,Y 468.15,Z 340.531,A -85,B 0,C 180,E1 -7471.936,E2 -7471.936} C_VEL
LIN {X 0,Y 467.605,Z 350.256,A -85,B 0,C 180,E1 -7473.231,E2 -7473.231} C_VEL
LIN {X 0,Y 467.279,Z 358.058,A -85,B 0,C 180,E1 -7474.529,E2 -7474.529} C_VEL
LIN {X 0,Y 467.058,Z 363.359,A -85,B 0,C 180,E1 -7475.613,E2 -7475.613} C_VEL
LIN {X 0,Y 466.914,Z 368.544,A -85,B 0,C 180,E1 -7476.916,E2 -7476.916} C_VEL
LIN {X 0,Y 466.793,Z 372.584,A -85,B 0,C 180,E1 -7478.223,E2 -7478.223} C_VEL
LIN {X 0,Y 466.626,Z 375.585,A -85,B 0,C 180,E1 -7479.536,E2 -7479.536} C_VEL
LIN {X 0,Y 466.63,Z 377.028,A -85,B 0,C 180,E1 -7480.412,E2 -7480.412} C_VEL
LIN {X 0,Y 466.633,Z 378.459,A -85,B 0,C 180,E1 -7481.779,E2 -7481.779} C_VEL
LIN {X 0,Y 466.545,Z 378.91,A -85,B 0,C 180,E1 -7483.059,E2 -7483.059} C_VEL
LIN {X 0,Y 466.517,Z 378.687,A -85,B 0,C 180,E1 -7483.947,E2 -7483.947} C_VEL
LIN {X 0,Y 466.603,Z 377.403,A -85,B 0,C 180,E1 -7485.433,E2 -7485.433} C_VEL
LIN {X 0,Y 466.595,Z 375.524,A -85,B 0,C 180,E1 -7486.629,E2 -7486.629} C_VEL
LIN {X 0,Y 466.782,Z 372.407,A -85,B 0,C 180,E1 -7487.978,E2 -7487.978} C_VEL
LIN {X 0,Y 466.921,Z 368.132,A -85,B 0,C 180,E1 -7489.337,E2 -7489.337} C_VEL
LIN {X 0,Y 467.125,Z 362.559,A -85,B 0,C 180,E1 -7490.705,E2 -7490.705} C_VEL
LIN {X 0,Y 467.481,Z 355.494,A -85,B 0,C 180,E1 -7492.076,E2 -7492.076} C_VEL
LIN {X 0,Y 467.905,Z 347.264,A -85,B 0,C 180,E1 -7493.355,E2 -7493.355} C_VEL
LIN {X 0,Y 468.34,Z 338.212,A -85,B 0,C 180,E1 -7494.49,E2 -7494.49} C_VEL
LIN {X 0,Y 468.854,Z 328.027,A -85,B 0,C 180,E1 -7495.528,E2 -7495.528} C_VEL
LIN {X 0,Y 469.378,Z 316.595,A -85,B 0,C 180,E1 -7496.459,E2 -7496.459} C_VEL
LIN {X 0,Y 469.866,Z 304.824,A -85,B 0,C 180,E1 -7497.202,E2 -7497.202} C_VEL
LIN {X 0,Y 470.311,Z 292.211,A -85,B 0,C 180,E1 -7497.801,E2 -7497.801} C_VEL
LIN {X 0,Y 467.983,Z 280.089,A -85,B 0,C 180,E1 -7498.301,E2 -7498.301} C_VEL
LIN {X 0,Y 466.796,Z 274.793,A -85,B 0,C 180,E1 -7498.496,E2 -7498.496} C_VEL
LIN {X 0,Y 466.879,Z 269.727,A -85,B 0,C 180,E1 -7501.793,E2 -7501.793} C_VEL
LIN {X 0,Y 467.008,Z 265.082,A -85,B 0,C 180,E1 -7504.879,E2 -7504.879} C_VEL
LIN {X 0,Y 467.142,Z 260.384,A -85,B 0,C 180,E1 -7508.084,E2 -7508.084} C_VEL
LIN {X 0,Y 467.234,Z 255.867,A -85,B 0,C 180,E1 -7511.231,E2 -7511.231} C_VEL
LIN {X 0,Y 467.407,Z 252.267,A -85,B 0,C 180,E1 -7513.804,E2 -7513.804} C_VEL
LIN {X 0,Y 467.535,Z 248.906,A -85,B 0,C 180,E1 -7516.255,E2 -7516.255} C_VEL
LIN {X 0,Y 467.535,Z 245.644,A -85,B 0,C 180,E1 -7518.728,E2 -7518.728} C_VEL
LIN {X 0,Y 467.55,Z 245.252,A -85,B 0,C 180,E1 -7520.049,E2 -7520.049} C_VEL
LIN {X 0,Y 467.52,Z 245.251,A -85,B 0,C 180,E1 -7523.039,E2 -7523.039} C_VEL
LIN {X 0,Y 467.573,Z 245.245,A -85,B 0,C 180,E1 -7526.212,E2 -7526.212} C_VEL
LIN {X 0,Y 467.561,Z 245.245,A -85,B 0,C 180,E1 -7529.267,E2 -7529.267} C_VEL
LIN {X 0,Y 467.621,Z 245.236,A -85,B 0,C 180,E1 -7532.462,E2 -7532.462} C_VEL
LIN {X 0,Y 467.593,Z 245.241,A -85,B 0,C 180,E1 -7535.113,E2 -7535.113} C_VEL
LIN {X 0,Y 467.563,Z 245.247,A -85,B 0,C 180,E1 -7537.929,E2 -7537.929} C_VEL
LIN {X 0,Y 467.612,Z 245.239,A -85,B 0,C 180,E1 -7540.693,E2 -7540.693} C_VEL
LIN {X 0,Y 467.655,Z 245.233,A -85,B 0,C 180,E1 -7544.108,E2 -7544.108} C_VEL
LIN {X 0,Y 467.644,Z 245.233,A -85,B 0,C 180,E1 -7547.855,E2 -7547.855} C_VEL
LIN {X 0,Y 467.672,Z 245.233,A -85,B 0,C 180,E1 -7551.358,E2 -7551.358} C_VEL
LIN {X 0,Y 467.72,Z 245.223,A -85,B 0,C 180,E1 -7553.963,E2 -7553.963} C_VEL
LIN {X 0,Y 467.851,Z 245.21,A -85,B 0,C 180,E1 -7557.418,E2 -7557.418} C_VEL
LIN {X 0,Y 467.868,Z 245.204,A -85,B 0,C 180,E1 -7560.001,E2 -7560.001} C_VEL
LIN {X 0,Y 467.852,Z 245.207,A -85,B 0,C 180,E1 -7562.584,E2 -7562.584} C_VEL
LIN {X 0,Y 467.725,Z 245.222,A -85,B 0,C 180,E1 -7566.039,E2 -7566.039} C_VEL
LIN {X 0,Y 467.673,Z 245.229,A -85,B 0,C 180,E1 -7568.644,E2 -7568.644} C_VEL
LIN {X 0,Y 467.649,Z 245.233,A -85,B 0,C 180,E1 -7572.147,E2 -7572.147} C_VEL
LIN {X 0,Y 467.631,Z 245.239,A -85,B 0,C 180,E1 -7575.696,E2 -7575.696} C_VEL
LIN {X 0,Y 467.61,Z 245.241,A -85,B 0,C 180,E1 -7578.766,E2 -7578.766} C_VEL
LIN {X 0,Y 467.573,Z 245.245,A -85,B 0,C 180,E1 -7581.269,E2 -7581.269} C_VEL
LIN {X 0,Y 467.567,Z 245.245,A -85,B 0,C 180,E1 -7583.944,E2 -7583.944} C_VEL
LIN {X 0,Y 467.565,Z 245.245,A -85,B 0,C 180,E1 -7586.804,E2 -7586.804} C_VEL
LIN {X 0,Y 467.542,Z 245.248,A -85,B 0,C 180,E1 -7589.74,E2 -7589.74} C_VEL
LIN {X 0,Y 467.579,Z 245.242,A -85,B 0,C 180,E1 -7592.76,E2 -7592.76} C_VEL
LIN {X 0,Y 467.549,Z 245.245,A -85,B 0,C 180,E1 -7595.891,E2 -7595.891} C_VEL
LIN {X 0,Y 467.579,Z 245.241,A -85,B 0,C 180,E1 -7599.146,E2 -7599.146} C_VEL
LIN {X 0,Y 467.584,Z 245.241,A -85,B 0,C 180,E1 -7602.568,E2 -7602.568} C_VEL
LIN {X 0,Y 467.563,Z 245.239,A -85,B 0,C 180,E1 -7605.054,E2 -7605.054} C_VEL
LIN {X 0,Y 467.561,Z 245.249,A -85,B 0,C 180,E1 -7608.727,E2 -7608.727} C_VEL
LIN {X 0,Y 467.595,Z 245.366,A -85,B 0,C 180,E1 -7610.3,E2 -7610.3} C_VEL
LIN {X 0,Y 468.418,Z 250.455,A -85,B 0,C 180,E1 -7613.121,E2 -7613.121} C_VEL
LIN {X 0,Y 468.612,Z 255.225,A -85,B 0,C 180,E1 -7615.575,E2 -7615.575} C_VEL
LIN {X 0,Y 468.236,Z 261.951,A -85,B 0,C 180,E1 -7618.821,E2 -7618.821} C_VEL
LIN {X 0,Y 467.881,Z 268.321,A -85,B 0,C 180,E1 -7621.761,E2 -7621.761} C_VEL
LIN {X 0,Y 467.56,Z 275.853,A -85,B 0,C 180,E1 -7625.111,E2 -7625.111} C_VEL
